No03: NOP   0;
NoXX: NOP   0;
NETWORK
TITLE =ASW_6030: Active step germinating
//      U     "MAL1S021Par".Par.FlagProcess.ProcessActive;
//      SPBN  tuen;
//
//// copy stepnr
//      L     "MAL1S021Par".Par.ParIntMachine.ActualStep;
//      T     "MAL1S021Par".Par.ParIntProcess.ActualStep;
//// set step conditions
//
//// Case where process is starting during loading
//      U     "MAL1S021Par".Par.FlagProcess.ProcessActive;
//      UN    "MAL1S021Par".Par.FlagFunction_1.StepLoading; // Step loading
//      SPBN  e003;
//// lifting devices must be in highest position
//      L       WinCoS_BIW01_09PLC1BIW01_02.Ma.Par.ParPositionTopRightUnits;
////Malting Plant OAO Belsolod Ivanonvo Weissrussland
//      L     50; // 50mm offset
//      +I    ;
//      T     "MAL1S021Par".Par.MachineValue.SOLLWERT_HUBZUG1_HOEHE;
//      L       WinCoS_BIW01_09PLC1BIW01_02.Ma.Par.ParPositionTopLeftUnits;
////Malting Plant OAO Belsolod Ivanonvo Weissrussland
//      L     50; // 50mm offset
//      +I    ;
//      T     "MAL1S021Par".Par.MachineValue.SOLLWERT_HUBZUG2_HOEHE;
//      L     5;
//      T     WinCoS_BIW01_09PLC1BIW01_02.Ma.Par.ParTolPosition;
//e003: NOP   0;
//
//// reset turning cmds
//
//// save turning cmds from prev.step
//      L     "MAL1S021Par".Par.ParIntMachine.ActualStep;
//      L     "MAL1S021Par".Par.ParIntProcess.PrevStep1stTurn;
//      <>I   ;
//      SPB   sav1;
//      U     "MAL1S021Par".Par.FlagProcess2.Turning1WithSpraying;
//      =     "MAL1S021Par".Par.Switches1.StaOn08; // Turning1WithSpraying
//      U     "MAL1S021Par".Par.FlagProcess2.Turning1WithDosing;
//      =     "MAL1S021Par".Par.Switches1.StaOn09; // Turning1WithDosing
//sav1: NOP   0;
//      L     "MAL1S021Par".Par.ParIntMachine.ActualStep;
//      L     "MAL1S021Par".Par.ParIntProcess.PrevStep2ndTurn;
//      <>I   ;
//      SPB   sav2;
//      U     "MAL1S021Par".Par.FlagProcess2.Turning2WithSpraying;
//      =     "MAL1S021Par".Par.Switches1.StaOn10; // Turning2WithSpraying
//      U     "MAL1S021Par".Par.FlagProcess2.Turning2WithDosing;
//      =     "MAL1S021Par".Par.Switches1.StaOn11; // Turning2WithDosing
//sav2: NOP   0;
//
//      SET   ;
//      R     "MAL1S021Par".Par.FlagProcess2.Turning1WithoutSpraying;
//      R     "MAL1S021Par".Par.FlagProcess2.Turning1WithSpraying;
//      R     "MAL1S021Par".Par.FlagProcess2.Turning1WithDosing;
//      R     "MAL1S021Par".Par.FlagProcess2.Turning2WithoutSpraying;
//      R     "MAL1S021Par".Par.FlagProcess2.Turning2WithSpraying;
//      R     "MAL1S021Par".Par.FlagProcess2.Turning2WithDosing;
//
//// Delta Temp to switch to next step
//      L     "MAL1S021Par".StepAct.DeltaTempSwitchpointStep;
//      L     L#0;
//      >D   ;
//      =     "MAL1S021Par".Par.FlagProcess1.DeltaTempNextStep;
//// Max Temp to switch to next step
//      L     "MAL1S021Par".StepAct.MaxTempAboveFloorStep;
//      L     L#0;
//      >D   ;
//      =     "MAL1S021Par".Par.FlagProcess1.MaxTempNextStep;
//
//// position waste air see sub 6050
//
//// basic speed fan see sub 6040
//
//// air humifidication
//      L     1;
//      L     "MAL1S021Par".StepAct.AirMoisten;   // On/Off
//      ==I;  // air humifidication on
//      U     WinCoS_BIW01_09PLC1BIW01_02.Ma.StStartedFwd; //Malting Plant OAO Be
//lsolod Ivanonvo Weissrussland
//      =     "MAL1S021Par".Par.FlagProcess.AirHumidificationValve1; // air humif
//idication valve 1 on
//      U(    ; // air humifidication on
//      L     "MAL1S021Par".Par.ParIntMachine.TargetSpeedGermFan; // germinating
//fan is running
//      L     40; // fanspeed > 40%
//      >I    ; // muss noch in Istwert getauscht werden JV
//      )     ; // fanspeed > 40%
//      =     "MAL1S021Par".Par.FlagProcess.AirHumidificationValve2;
//
//// air cooling
//      L     "MAL1S021Par".StepAct.Cooling;
//      L   1;  // Activate Cooling System = 1 (yes)
//      ==I;
//      =     "MAL1S021Par".Par.FlagProcess.Cooling; // request cooling
//
//      U     "MAL1S021Par".Par.FlagProcess.ProcessActive;
//      U     "MAL1S021".PCRead.Step.StReady;
//      UN    "MAL1S021Par".Par.FlagFunction_1.StepLoading;
//      SPBN  e630;
//
//// turning 1
//      UN    "MAL1S021Par".Par.FlagProcess2.StartSecondTurningRound; // Turn
//from PrevStep
//      U(;
//      L     "MAL1S021Par".StepAct.StartTurningRound_1;
//      L     0;
//      >=D;                  // negative, no turning 1
//      );
//      U(    ;
//      O(    ; // Nach Rezept
//      L     "MAL1S021Par".ActTimeStepProcess.StepTimeActHourTotal; // Steptime
//in hours overall
//      L     "MAL1S021Par".StepAct.StartTurningRound_1;
//      ==I   ;
//      UN     WinCoS_BIW01_09PLC1BIW01_02.Ma.StAdjusted; // target position
//turning reached
//      )     ;
//      O(    ; // Selbsthaltung
//      L     "MAL1S021Par".ActTimeStepProcess.StepTimeActHourTotal; // Steptime i
//n hours overall
//      L     "MAL1S021Par".StepAct.StartTurningRound_1;
//      <>I   ;
//      U     "MAL1S021Par".Par.FlagProcess2.StartFirstTurningRound;
//      )     ;
//      )     ;
//      S     "MAL1S021Par".Par.FlagProcess2.Turning1WithoutSpraying;
//      S     "MAL1S021Par".Par.FlagFunction_1.TurningStart;
//// turning 1 with spraying
//      U(    ;
//      L     1;
//      L     "MAL1S021Par".StepAct.TurningWithSpraying_1;
//      ==I;    // turning 1 with spraying on
//      U(    ;
//      L     "MAL1S021Par".Par.ParIntMachine.ActualStep;
//      L     "MAL1S021Par".Par.ParIntProcess.PrevStep1stTurn;
//      ==I   ;
//      )     ;
//      )     ;
//      O(    ;
//      L     "MAL1S021Par".Par.ParIntMachine.ActualStep;
//      L     "MAL1S021Par".Par.ParIntProcess.PrevStep1stTurn;
//      <>I   ;
//      U     "MAL1S021Par".Par.Switches1.StaOn08; // Turning1WithSpraying
//      )     ;
//      U     "MAL1S021Par".Par.FlagProcess2.Turning1WithoutSpraying;
//      S     "MAL1S021Par".Par.FlagProcess2.Turning1WithSpraying;
//// turning 1 with spraying and GA3
//      U(    ;
//      L     1;
//      L     "MAL1S021Par".StepAct.TurningWithDosing_1;
//      ==I;    // turning 1 with spraying on
//      U(    ;
//      L     "MAL1S021Par".Par.ParIntMachine.ActualStep;
//      L     "MAL1S021Par".Par.ParIntProcess.PrevStep1stTurn;
//      ==I   ;
//      )     ;
//      )     ;
//      O(    ;
//      L     "MAL1S021Par".Par.ParIntMachine.ActualStep;
//      L     "MAL1S021Par".Par.ParIntProcess.PrevStep1stTurn;
//      <>I   ;
//      U     "MAL1S021Par".Par.Switches1.StaOn09; // Turning1WithDosing
//      )     ;
//      U     "MAL1S021Par".Par.FlagProcess2.Turning1WithoutSpraying;
//      S     "MAL1S021Par".Par.FlagProcess2.Turning1WithSpraying;
//      S     "MAL1S021Par".Par.FlagProcess2.Turning1WithDosing;
//
//      U     "MAL1S021Par".Par.FlagProcess2.Turning1WithoutSpraying;
//      U     "MAL1S021Par".Par.FlagFunction_1.TurningStart;
//      UN     WinCoS_BIW01_09PLC1BIW01_02.Ma.StAdjusted; // target position turni
//ng reached
//      FP    "MAL1S021Par".Par.FlagProcess2.StartFirstTurningFP;
//      S     "MAL1S021Par".Par.FlagProcess2.StartFirstTurningRound;
//
//      U     WinCoS_BIW01_09PLC1BIW01_02.Ma.StAdjusted; // target position
//turning reached
//      O(    ;
//      L     "MAL1S021Par".ActTimeStepProcess.StepTimeActHourTotal; // Steptime i
//n hours overall
//      L     "MAL1S021Par".StepAct.StartTurningRound_1;
//      >I    ;
//      U     WinCoS_BIW01_09PLC1BIW01_02.Ma.StAdjusted; // target position
//turning reached
//      )     ;
//      U     "MAL1S021Par".Par.FlagProcess2.StartFirstTurningRound;
//      R     "MAL1S021Par".Par.FlagProcess2.StartFirstTurningRound;
//
//      U     "MAL1S021Par".Par.FlagProcess2.StartFirstTurningFP;
//      SPB   trn1;
//      L     "MAL1S021Par".Par.ParIntMachine.ActualStep;
//      T     "MAL1S021Par".Par.ParIntProcess.PrevStep1stTurn;
//trn1: NOP   0;
//
//// turning 2
//      UN    "MAL1S021Par".Par.FlagProcess2.StartFirstTurningRound; // Unsinngie
//Rezeptwerte
//      U(;
//      L     1;
//      L     "MAL1S021Par".StepAct.StartTurningRound_2;
//      ==I    ;
//      );
//      U(    ;
//      O(    ; // Nach Rezept
//      L     "MAL1S021Par".ActTimeStepProcess.StepTimeActHourTotal; // Steptime i
//n hours overall
//      L     "MAL1S021Par".StepAct.StartTurningRound_2;
//      ==I   ;
//      UN     WinCoS_BIW01_09PLC1BIW01_02.Ma.StAdjusted; // target position
//turning reached
//      )     ;
//      O(    ; // Selbsthaltung
//      L     "MAL1S021Par".ActTimeStepProcess.StepTimeActHourTotal; // Steptime
//in hours overall
//      L     "MAL1S021Par".StepAct.StartTurningRound_2;
//      <>I   ;
//      U     "MAL1S021Par".Par.FlagProcess2.StartSecondTurningRound;
//      )     ;
//      )     ;
//      S     "MAL1S021Par".Par.FlagProcess2.Turning2WithoutSpraying;
//      S     "MAL1S021Par".Par.FlagFunction_1.TurningStart;
//// turning 2 with spraying
//      U(    ;
//      L     1;
//      L     "MAL1S021Par".StepAct.TurningWithSpraying_2;
//      ==I    ;
//      U(    ;
//      L     "MAL1S021Par".Par.ParIntMachine.ActualStep;
//      L     "MAL1S021Par".Par.ParIntProcess.PrevStep2ndTurn;
//      ==I   ;
//      )     ;
//      )     ;
//      O(    ;
//      L     "MAL1S021Par".Par.ParIntMachine.ActualStep;
//      L     "MAL1S021Par".Par.ParIntProcess.PrevStep2ndTurn;
//      <>I   ;
//      U     "MAL1S021Par".Par.Switches1.StaOn10; // Turning2WithSpraying
//      )     ;
//      U     "MAL1S021Par".Par.FlagProcess2.Turning2WithoutSpraying;
//      S     "MAL1S021Par".Par.FlagProcess2.Turning2WithSpraying;
//// turning 2 with spraying and GA3
//      U(    ;
//      L     1;
//      L     "MAL1S021Par".StepAct.TurningWithDosing_2;
//      ==I;    // turning 2 with spraying and GA3 on
//      U(    ;
//      L     "MAL1S021Par".Par.ParIntMachine.ActualStep;
//      L     "MAL1S021Par".Par.ParIntProcess.PrevStep2ndTurn;
//      ==I   ;
//      )     ;
//      )     ;
//      O(    ;
//      L     "MAL1S021Par".Par.ParIntMachine.ActualStep;
//      L     "MAL1S021Par".Par.ParIntProcess.PrevStep2ndTurn;
//      <>I   ;
//      U     "MAL1S021Par".Par.Switches1.StaOn11; // Turning2WithDosing
//      )     ;
//      U     "MAL1S021Par".Par.FlagProcess2.Turning2WithoutSpraying;
//      S     "MAL1S021Par".Par.FlagProcess2.Turning2WithSpraying;
//      S     "MAL1S021Par".Par.FlagProcess2.Turning2WithDosing;
//
//      U     "MAL1S021Par".Par.FlagProcess2.Turning2WithoutSpraying;
//      U     "MAL1S021Par".Par.FlagFunction_1.TurningStart;
//      UN     WinCoS_BIW01_09PLC1BIW01_02.Ma.StAdjusted; // target position
//turning reached
//      FP    "MAL1S021Par".Par.FlagProcess2.StartSecondTurningFP;
//      S     "MAL1S021Par".Par.FlagProcess2.StartSecondTurningRound;
//
//      U     WinCoS_BIW01_09PLC1BIW01_02.Ma.StAdjusted; // target position
//turning reached
//      O(    ;
//      L     "MAL1S021Par".ActTimeStepProcess.StepTimeActHourTotal; // Steptime
//in hours overall
//      L     "MAL1S021Par".StepAct.StartTurningRound_2;
//      >I    ;
//      U     WinCoS_BIW01_09PLC1BIW01_02.Ma.StAdjusted; // target position
//turning reached
//      )     ;
//      U     "MAL1S021Par".Par.FlagProcess2.StartSecondTurningRound;
//      R     "MAL1S021Par".Par.FlagProcess2.StartSecondTurningRound;
//
//      U     "MAL1S021Par".Par.FlagProcess2.StartSecondTurningFP;
//      SPB   trn2;
//      L     "MAL1S021Par".Par.ParIntMachine.ActualStep;
//      T     "MAL1S021Par".Par.ParIntProcess.PrevStep2ndTurn;
//trn2: NOP   0;
////Fix Speed for Turning
//      U     "MAL1S021Par".Par.FlagProcess2.Turning1WithoutSpraying;
//      O     "MAL1S021Par".Par.FlagProcess2.Turning1WithSpraying;
//      O     "MAL1S021Par".Par.FlagProcess2.Turning2WithoutSpraying;
//      O     "MAL1S021Par".Par.FlagProcess2.Turning2WithSpraying;
//      U    M 50.0;
//      SPBN  SpdT;
//      L     15; // 15Hz
//      T     "MAL1S021Par".Par.MachineValue.SollwertFahrantrieb;
//SpdT: NOP   0;
//
//// find turning direction
//      U     "MAL1S021Par".Par.FlagGen.TurningStarted;
//      O(    ;
//      UN    "MAL1S021Par".Par.FlagProcess2.Turning1WithoutSpraying;
//      UN    "MAL1S021Par".Par.FlagProcess2.Turning2WithoutSpraying;
//      )     ;
//      SPB   tuen;
//      L     "MAL1S021Par".Par.ParIntMachine.TargetPosTravDriTurnRigt; // 370° =
//endposition turning right
//      T     WinCoS_BIW01_09PLC1BIW01_02.Ma.InPositionTarget; // target position
//turning reached
//
//      U(    ;
//      L     WinCoS_BIW01_09PLC1BIW01_02.Ma.OutPositionAngle;
//      L     1800;
//      <I    ; // condition turning right (clockwise)
//      )     ;
//      S     "MAL1S021Par".Par.FlagFunction_1.TurningRight;
//      S     "MAL1S021Par".Par.FlagGen.TurningStarted;
//// - Correct effect of ILO Mode
//      L       WinCoS_BIW01_09PLC1BIW01_02.Ma.Par.ParPositionTopLeftUnits; //Malt
//ing Plant OAO Belsolod Ivanonvo Weissrussland
//      T     "MAL1S021Par".Par.MachineValue.SOLLWERT_HUBZUG1_HOEHE;
//      L       WinCoS_BIW01_09PLC1BIW01_02.Ma.Par.ParPositionTopRightUnits; //Mal
//ting Plant OAO Belsolod Ivanonvo Weissrussland
//      T     "MAL1S021Par".Par.MachineValue.SOLLWERT_HUBZUG2_HOEHE;
//      SPB   E603   ;
//      L     "MAL1S021Par".Par.ParIntMachine.TargetPosTravDriTurnLeft; // 0° =
//endposition turning left
//      T     WinCoS_BIW01_09PLC1BIW01_02.Ma.InPositionTarget; // target position
//turning reached
//
//      U(    ;
//      L     WinCoS_BIW01_09PLC1BIW01_02.Ma.OutPositionAngle;
//      L     1800;
//      >=I   ; // condition turning left (counterclockwise)
//      )     ;
//      S     "MAL1S021Par".Par.FlagFunction_1.TurningLeft;
//      S     "MAL1S021Par".Par.FlagGen.TurningStarted;
//// - Correct effect of ILO Mode
//      L       WinCoS_BIW01_09PLC1BIW01_02.Ma.Par.ParPositionTopLeftUnits;
////Malting Plant OAO Belsolod Ivanonvo Weissrussland
//      T     "MAL1S021Par".Par.MachineValue.SOLLWERT_HUBZUG1_HOEHE;
//      L       WinCoS_BIW01_09PLC1BIW01_02.Ma.Par.ParPositionTopRightUnits;
////Malting Plant OAO Belsolod Ivanonvo Weissrussland
//      T     "MAL1S021Par".Par.MachineValue.SOLLWERT_HUBZUG2_HOEHE;
//      SPB   E603   ;
//tuen: NOP   0;
//// - Case of fast speed to protect a 2nd start during same hours as finsihed
//      O(    ; // Nach Rezept
//      L     "MAL1S021Par".ActTimeStepProcess.StepTimeActHourTotal; // Steptime i
//n hours overall
//      L     "MAL1S021Par".StepAct.StartTurningRound_1;
//      ==I   ;
//      U     WinCoS_BIW01_09PLC1BIW01_02.Ma.StAdjusted; // target position turnin
//g reached
//      U     "MAL1S021Par".Par.FlagFunction_1.TurningStart;
//      )     ;
//      O(    ; // Nach Rezept
//      L     "MAL1S021Par".ActTimeStepProcess.StepTimeActHourTotal; // Steptime i
//n hours overall
//      L     "MAL1S021Par".StepAct.StartTurningRound_2;
//      ==I   ;
//      U     WinCoS_BIW01_09PLC1BIW01_02.Ma.StAdjusted; // target position
//turning reached
//      U     "MAL1S021Par".Par.FlagFunction_1.TurningStart;
//      )     ;
//      SPB   e603;
//
//// reset turning right (clockwise)
//      U     "MAL1S021Par".Par.FlagFunction_1.TurningRight;
//      U(    ;
//      O      WinCoS_BIW01_09PLC1BIW01_02.Ma.StAdjusted; // target position
//turning reached
//      O(    ;
//      L     WinCoS_BIW01_09PLC1BIW01_02.Ma.OutPositionAngle;
//      L     WinCoS_BIW01_09PLC1BIW01_02.Ma.Par.ParTolPosition;
//      +I    ;
//      L     "MAL1S021Par".Par.ParIntMachine.TargetPosTravDriTurnRigt;
//      >=I   ;
//      )     ;
//      )     ;
//      R     "MAL1S021Par".Par.FlagFunction_1.TurningRight;
//      R     "MAL1S021Par".Par.FlagFunction_1.TurningStart;
//
//// reset turning left (counterclockwise)
//      U     "MAL1S021Par".Par.FlagFunction_1.TurningLeft;
//      U(    ;
//      O     WinCoS_BIW01_09PLC1BIW01_02.Ma.StAdjusted; // target position turnin
//g reached
//      O(    ;
//      L     WinCoS_BIW01_09PLC1BIW01_02.Ma.OutPositionAngle;
//      L     WinCoS_BIW01_09PLC1BIW01_02.Ma.Par.ParTolPosition;
//      -I    ;
//      L     "MAL1S021Par".Par.ParIntMachine.TargetPosTravDriTurnLeft;
//      <=I   ;
//      )     ;
//      )     ;
//      R     "MAL1S021Par".Par.FlagFunction_1.TurningLeft;
//      R     "MAL1S021Par".Par.FlagFunction_1.TurningStart;
//
//// reset turning flag
//      U     "MAL1S021Par".Par.FlagGen.TurningStarted;
//      UN    "MAL1S021Par".Par.FlagProcess2.Turning1WithoutSpraying;
//      UN    "MAL1S021Par".Par.FlagProcess2.Turning2WithoutSpraying;
//      O(    ;
//      U     "MAL1S021Par".Par.FlagGen.TurningStarted;
//      U     WinCoS_BIW01_09PLC1BIW01_02.Ma.StAdjusted; // target position
//turning reached
//      )     ;
//      ON    "MAL1S021Par".Par.FlagProcess.ProcessActive;
//      R     "MAL1S021Par".Par.FlagGen.TurningStarted;
//      R     "MAL1S021Par".Par.FlagProcess2.Turning1WithoutSpraying;
//      R     "MAL1S021Par".Par.FlagProcess2.Turning2WithoutSpraying;
//      R     "MAL1S021Par".Par.FlagFunction_1.TurningStart;
//e630: NOP   0;
//      UN    "MAL1S021Par".Par.FlagProcess.ProcessActive;
//      R     "MAL1S021Par".Par.FlagProcess2.StartFirstTurningRound;
//      R     "MAL1S021Par".Par.FlagProcess2.StartSecondTurningRound;
//
//e603: NOP   0;
//E603: NOP   0;



      U     "MAL1S021Par".Par.FlagProcess.ProcessActive;
      SPBN  tuen;

// copy stepnr
      L     "MAL1S021Par".Par.ParIntMachine.ActualStep;
      T     "MAL1S021Par".Par.ParIntProcess.ActualStep;
// set step conditions

// reset turning cmds

// save turning cmds from prev.step
      L     "MAL1S021Par".Par.ParIntMachine.ActualStep;
      L     "MAL1S021Par".Par.ParIntProcess.PrevStep1stTurn;
      <>I   ;
      SPB   sav1;
      U     "MAL1S021Par".Par.FlagProcess2.Turning1WithSpraying;
      =     "MAL1S021Par".Par.Switches1.StaOn08; // Turning1WithSpraying
      U     "MAL1S021Par".Par.FlagProcess2.Turning1WithDosing;
      =     "MAL1S021Par".Par.Switches1.StaOn09; // Turning1WithDosing
sav1: NOP   0;
      L     "MAL1S021Par".Par.ParIntMachine.ActualStep;
      L     "MAL1S021Par".Par.ParIntProcess.PrevStep2ndTurn;
      <>I   ;
      SPB   sav2;
      U     "MAL1S021Par".Par.FlagProcess2.Turning2WithSpraying;
      =     "MAL1S021Par".Par.Switches1.StaOn10; // Turning2WithSpraying
      U     "MAL1S021Par".Par.FlagProcess2.Turning2WithDosing;
      =     "MAL1S021Par".Par.Switches1.StaOn11; // Turning2WithDosing
sav2: NOP   0;

      SET   ;
      R     "MAL1S021Par".Par.FlagProcess2.Turning1WithoutSpraying;
      R     "MAL1S021Par".Par.FlagProcess2.Turning1WithSpraying;
      R     "MAL1S021Par".Par.FlagProcess2.Turning1WithDosing;
      R     "MAL1S021Par".Par.FlagProcess2.Turning2WithoutSpraying;
      R     "MAL1S021Par".Par.FlagProcess2.Turning2WithSpraying;
      R     "MAL1S021Par".Par.FlagProcess2.Turning2WithDosing;

// Delta Temp to switch to next step
      L     "MAL1S021Par".StepAct.DeltaTempSwitchpointStep;
      L     L#0;
      >D    ;
      =     "MAL1S021Par".Par.FlagProcess1.DeltaTempNextStep;
// Max Temp to switch to next step
      L     "MAL1S021Par".StepAct.MaxTempAboveFloorStep;
      L     L#0;
      >D    ;
      =     "MAL1S021Par".Par.FlagProcess1.MaxTempNextStep;

// position waste air see sub 6050

// basic speed fan see sub 6040

// air humifidication

// air cooling
      L     "MAL1S021Par".StepAct.Cooling;
      L     1; // Activate Cooling System = 1 (yes)
      ==I   ;
      =     "MAL1S021Par".Par.FlagProcess.Cooling; // request cooling

      U     "MAL1S021Par".Par.FlagProcess.ProcessActive;
      U     "MAL1S021".PCRead.Step.StReady;
      UN    "MAL1S021Par".Par.FlagFunction_1.StepLoading;
      SPBN  e630;

// turning 1
      UN    "MAL1S021Par".Par.FlagProcess2.StartSecondTurningRound; // Turn from PrevStep
      U(    ;
      L     "MAL1S021Par".StepAct.StartTurningRound_1;
      L     0;
      >=I   ; // negative, no turning 1
      )     ;
      U(    ;
      O(    ; // Nach Rezept
      L     "MAL1S021Par".ActTimeStepProcess.StepTimeActHourTotal; // Steptime in hours overall
      L     "MAL1S021Par".StepAct.StartTurningRound_1;
      ==I   ;
      UN    "G185M".A_2511_MXZ41MA.Ma.StAdjusted; // target position turning reached
      )     ;
      O(    ; // Selbsthaltung
      L     "MAL1S021Par".ActTimeStepProcess.StepTimeActHourTotal; // Steptime in hours overall
      L     "MAL1S021Par".StepAct.StartTurningRound_1;
      <>I   ;
      U     "MAL1S021Par".Par.FlagProcess2.StartFirstTurningRound;
      )     ;
      )     ;
      S     "MAL1S021Par".Par.FlagProcess2.Turning1WithoutSpraying;
      S     "MAL1S021Par".Par.FlagFunction_1.TurningStart;
// turning 1 with spraying
      U(    ;
      L     1;
      L     "MAL1S021Par".StepAct.TurningWithSpraying_1;
      ==I   ; // turning 1 with spraying on
      U(    ;
      L     "MAL1S021Par".Par.ParIntMachine.ActualStep;
      L     "MAL1S021Par".Par.ParIntProcess.PrevStep1stTurn;
      ==I   ;
      )     ;
      )     ;
      O(    ;
      L     "MAL1S021Par".Par.ParIntMachine.ActualStep;
      L     "MAL1S021Par".Par.ParIntProcess.PrevStep1stTurn;
      <>I   ;
      U     "MAL1S021Par".Par.Switches1.StaOn08; // Turning1WithSpraying
      )     ;
      U     "MAL1S021Par".Par.FlagProcess2.Turning1WithoutSpraying;
      S     "MAL1S021Par".Par.FlagProcess2.Turning1WithSpraying;
// turning 1 with spraying and GA3
      U(    ;
      L     1;
      L     "MAL1S021Par".StepAct.TurningWithDosing_1;
      ==I   ; // turning 1 with spraying on
      U(    ;
      L     "MAL1S021Par".Par.ParIntMachine.ActualStep;
      L     "MAL1S021Par".Par.ParIntProcess.PrevStep1stTurn;
      ==I   ;
      )     ;
      )     ;
      O(    ;
      L     "MAL1S021Par".Par.ParIntMachine.ActualStep;
      L     "MAL1S021Par".Par.ParIntProcess.PrevStep1stTurn;
      <>I   ;
      U     "MAL1S021Par".Par.Switches1.StaOn09; // Turning1WithDosing
      )     ;
      U     "MAL1S021Par".Par.FlagProcess2.Turning1WithoutSpraying;
      S     "MAL1S021Par".Par.FlagProcess2.Turning1WithSpraying;
      S     "MAL1S021Par".Par.FlagProcess2.Turning1WithDosing;

//BRT070410 - wird einen Zyklus später gesetzt
      U     "MAL1S021Par".Par.FlagProcess2.StartFirstDosingFP;
      S     "MAL1S021Par".Par.FlagProcess2.StartFirstTurningRound;

      U     "MAL1S021Par".Par.FlagProcess2.Turning1WithoutSpraying;
      U     "MAL1S021Par".Par.FlagFunction_1.TurningStart;
//BRT140310      UN    "G185M".A_2511_MXZ41MA.Ma.StAdjusted    // target position turning reached
      UN    "G185M".A_2511_MXZ41MA.Ma.OutAdjusted; // target position turning reached
      FP    "MAL1S021Par".Par.FlagProcess2.StartFirstTurningFP;
      =     "MAL1S021Par".Par.FlagProcess2.StartFirstDosingFP;
//BRT070410      S     "MAL1S021Par".Par.FlagProcess2.StartFirstTurningRound

      U     "MAL1S021Par".Par.FlagProcess2.StartFirstDosingFP;
      U     "MAL1S021Par".Par.FlagProcess2.StartFirstTurningFP;
      SPBN  trn1;
      L     "MAL1S021Par".Par.ParIntMachine.ActualStep;
      T     "MAL1S021Par".Par.ParIntProcess.PrevStep1stTurn;
trn1: NOP   0;

//BRT140310      U     "G185M".A_2511_MXZ41MA.Ma.StAdjusted    // target position turning reached
      U     "G185M".A_2511_MXZ41MA.Ma.OutAdjusted; // target position turning reached
      O(    ;
      L     "MAL1S021Par".ActTimeStepProcess.StepTimeActHourTotal; // Steptime in hours overall
      L     "MAL1S021Par".StepAct.StartTurningRound_1;
      >I    ;
      U(    ;
      O     "G185M".A_2511_MXZ41MA.Ma.OutAdjusted; // target position turning reached
      O(    ;
//BRT140310      UN    "G185M".A_2511_BZS46.StTrue // stop fan side
//BRT140310      U     "G185M".A_2511_BZS44.StTrue // stop discharge side
      U     "G185M".A_2511_BZS46.StTrue; // stop fan side
      UN    "G185M".A_2511_BZS44.StTrue; // stop discharge side
      U     "MAL1S021Par".Par.FlagFunction_1.TurningRight;
      )     ;
      O(    ;
//BRT140310      U     "G185M".A_2511_BZS46.StTrue // stop fan side
//BRT140310      UN    "G185M".A_2511_BZS44.StTrue // stop discharge side
      UN    "G185M".A_2511_BZS46.StTrue; // stop fan side
      U     "G185M".A_2511_BZS44.StTrue; // stop discharge side
      U     "MAL1S021Par".Par.FlagFunction_1.TurningLeft;
      )     ;
      )     ;
      )     ;
      O(    ;
      L     "MAL1S021Par".StepAct.StartTurningRound_1;
//BRT140310      L     0
//BRT140310      <D                                // negative, no turning 1
      L     -1; //BRT140310
      ==I   ; //BRT140310
      )     ;
      U     "MAL1S021Par".Par.FlagProcess2.StartFirstTurningRound;
      R     "MAL1S021Par".Par.FlagProcess2.StartFirstTurningRound;
      R     "MAL1S021Par".Par.Switches1.StaOn08; // Turning1WithSpraying
      R     "MAL1S021Par".Par.Switches1.StaOn09; // Turning1WithDosing

// turning 2
      UN    "MAL1S021Par".Par.FlagProcess2.StartFirstTurningRound; // Unsinnige Rezeptwerte
      U(    ;
//BRT160310      L     1
      L     "MAL1S021Par".StepAct.StartTurningRound_2;
      L     0; //BRT160310
      >=I   ;
      )     ;
      U(    ;
      O(    ; // Nach Rezept
      L     "MAL1S021Par".ActTimeStepProcess.StepTimeActHourTotal; // Steptime in hours overall
      L     "MAL1S021Par".StepAct.StartTurningRound_2;
      ==I   ;
      UN    "G185M".A_2511_MXZ41MA.Ma.StAdjusted; // target position turning reached
      )     ;
      O(    ; // Selbsthaltung
      L     "MAL1S021Par".ActTimeStepProcess.StepTimeActHourTotal; // Steptime in hours overall
      L     "MAL1S021Par".StepAct.StartTurningRound_2;
      <>I   ;
      U     "MAL1S021Par".Par.FlagProcess2.StartSecondTurningRound;
      )     ;
      )     ;
      S     "MAL1S021Par".Par.FlagProcess2.Turning2WithoutSpraying;
      S     "MAL1S021Par".Par.FlagFunction_1.TurningStart;
// turning 2 with spraying
      U(    ;
      L     1;
      L     "MAL1S021Par".StepAct.TurningWithSpraying_2;
      ==I   ;
      U(    ;
      L     "MAL1S021Par".Par.ParIntMachine.ActualStep;
      L     "MAL1S021Par".Par.ParIntProcess.PrevStep2ndTurn;
      ==I   ;
      )     ;
      )     ;
      O(    ;
      L     "MAL1S021Par".Par.ParIntMachine.ActualStep;
      L     "MAL1S021Par".Par.ParIntProcess.PrevStep2ndTurn;
      <>I   ;
      U     "MAL1S021Par".Par.Switches1.StaOn10; // Turning2WithSpraying
      )     ;
      U     "MAL1S021Par".Par.FlagProcess2.Turning2WithoutSpraying;
      S     "MAL1S021Par".Par.FlagProcess2.Turning2WithSpraying;
// turning 2 with spraying and GA3
      U(    ;
      L     1;
      L     "MAL1S021Par".StepAct.TurningWithDosing_2;
      ==I   ; // turning 2 with spraying and GA3 on
      U(    ;
      L     "MAL1S021Par".Par.ParIntMachine.ActualStep;
      L     "MAL1S021Par".Par.ParIntProcess.PrevStep2ndTurn;
      ==I   ;
      )     ;
      )     ;
      O(    ;
      L     "MAL1S021Par".Par.ParIntMachine.ActualStep;
      L     "MAL1S021Par".Par.ParIntProcess.PrevStep2ndTurn;
      <>I   ;
      U     "MAL1S021Par".Par.Switches1.StaOn11; // Turning2WithDosing
      )     ;
      U     "MAL1S021Par".Par.FlagProcess2.Turning2WithoutSpraying;
      S     "MAL1S021Par".Par.FlagProcess2.Turning2WithSpraying;
      S     "MAL1S021Par".Par.FlagProcess2.Turning2WithDosing;

//BRT070410 - wird einen Zyklus später gesetzt
      U     "MAL1S021Par".Par.FlagProcess2.StartSecondDosingFP;
      S     "MAL1S021Par".Par.FlagProcess2.StartSecondTurningRound;

      U     "MAL1S021Par".Par.FlagProcess2.Turning2WithoutSpraying;
      U     "MAL1S021Par".Par.FlagFunction_1.TurningStart;
//BRT140310      UN    "G185M".A_2511_MXZ41MA.Ma.StAdjusted    // target position turning reached
      UN    "G185M".A_2511_MXZ41MA.Ma.OutAdjusted; // target position turning reached
      FP    "MAL1S021Par".Par.FlagProcess2.StartSecondTurningFP;
      =     "MAL1S021Par".Par.FlagProcess2.StartSecondDosingFP;
//BRT070410      S     "MAL1S021Par".Par.FlagProcess2.StartSecondTurningRound

      U     "MAL1S021Par".Par.FlagProcess2.StartSecondDosingFP;
      U     "MAL1S021Par".Par.FlagProcess2.StartSecondTurningFP;
      SPBN  trn2;
      L     "MAL1S021Par".Par.ParIntMachine.ActualStep;
      T     "MAL1S021Par".Par.ParIntProcess.PrevStep2ndTurn;
trn2: NOP   0;

//BRT140310      U     "G185M".A_2511_MXZ41MA.Ma.StAdjusted    // target position turning reached
      U     "G185M".A_2511_MXZ41MA.Ma.OutAdjusted; // target position turning reached
      O(    ;
      L     "MAL1S021Par".ActTimeStepProcess.StepTimeActHourTotal; // Steptime in hours overall
      L     "MAL1S021Par".StepAct.StartTurningRound_2;
      >I    ;
      U(    ;
      O     "G185M".A_2511_MXZ41MA.Ma.OutAdjusted; // target position turning reached
      O(    ;
      UN    "G185M".A_2511_BZS46.StTrue; // stop fan side
      U     "G185M".A_2511_BZS44.StTrue; // stop discharge side
      U     "MAL1S021Par".Par.FlagFunction_1.TurningRight;
      )     ;
      O(    ;
      U     "G185M".A_2511_BZS46.StTrue; // stop fan side
      UN    "G185M".A_2511_BZS44.StTrue; // stop discharge side
      U     "MAL1S021Par".Par.FlagFunction_1.TurningLeft;
      )     ;
      )     ;
      )     ;
      O(    ;
      L     "MAL1S021Par".StepAct.StartTurningRound_2;
//BRT140310      L     0
//BRT140310      <D                                // negative, no turning 1
      L     -1; //BRT140310
      ==I   ; //BRT140310
      )     ;
      U     "MAL1S021Par".Par.FlagProcess2.StartSecondTurningRound;
      R     "MAL1S021Par".Par.FlagProcess2.StartSecondTurningRound;
      R     "MAL1S021Par".Par.Switches1.StaOn10; // Turning2WithSpraying
      R     "MAL1S021Par".Par.Switches1.StaOn11; // Turning2WithDosing

      L     3600;
      T     "MAL1S021Par".Par.ParIntMachine.TargetPosTravDriTurnRigt; // 360° = endposition turning right

// find turning direction spez. APU: right ==> forward, left ==> reverse
      U     "MAL1S021Par".Par.FlagGen.TurningStarted;
      O(    ;
      UN    "MAL1S021Par".Par.FlagProcess2.Turning1WithoutSpraying;
      UN    "MAL1S021Par".Par.FlagProcess2.Turning2WithoutSpraying;
      )     ;
      SPB   tuen;
      L     "MAL1S021Par".Par.ParIntMachine.TargetPosTravDriTurnRigt; // 360° = endposition turning right
      T     "G185M".A_2511_MXZ41MA.Ma.InPositionTarget; // target position turning

      U(    ;
      L     "G185M".A_2511_MXZ41MA.Ma.OutPositionAngle;
      L     1800;
      <I    ; // condition turning right (clockwise)
      )     ;
//BRT140310      O     "G185M".A_2511_BZS46.StTrue // stop fan side
//BRT140310      UN    "G185M".A_2511_BZS44.StTrue // stop discharge side
      O     "G185M".A_2511_BZS44.StTrue; // stop zeroposition  //BRT070310
      UN    "G185M".A_2511_BZS46.StTrue; //stop end side   //BRT070310
      S     "MAL1S021Par".Par.FlagFunction_1.TurningRight;
      S     "MAL1S021Par".Par.FlagGen.TurningStarted;
      SPB   E603;
      L     "MAL1S021Par".Par.ParIntMachine.TargetPosTravDriTurnLeft; // 0° = endposition turning left
      T     "G185M".A_2511_MXZ41MA.Ma.InPositionTarget; // target position turning

      U(    ;
      L     "G185M".A_2511_MXZ41MA.Ma.OutPositionAngle;
      L     1800;
      >=I   ; // condition turning left (counterclockwise)
      )     ;
//BRT140310      O     "G185M".A_2511_BZS44.StTrue // stop discharge side
//BRT140310      UN    "G185M".A_2511_BZS46.StTrue // stop fan side
      O     "G185M".A_2511_BZS46.StTrue; // stop zeroposition  //BRT070310
      UN    "G185M".A_2511_BZS44.StTrue; //stop end side   //BRT070310
      S     "MAL1S021Par".Par.FlagFunction_1.TurningLeft;
      S     "MAL1S021Par".Par.FlagGen.TurningStarted;
      SPB   E603;
tuen: NOP   0;

// reset turning right (clockwise)
      U     "MAL1S021Par".Par.FlagFunction_1.TurningRight;
      U(    ;
//      O     "G202M"._2111_MXZ41MA.Ma.StAdjusted    // target position turning reached
      O(    ;
      L     "G185M".A_2511_MXZ41MA.Ma.OutPositionAngle;
      L     "G185M".A_2511_MXZ41MA.Ma.Par.ParTolPosition;
      +I    ;
      L     "MAL1S021Par".Par.ParIntMachine.TargetPosTravDriTurnRigt;
      >=I   ;
      )     ;
//BRT140310      O     "G185M".A_2511_BZS44.StTrue // stop discharge side
      O     "G185M".A_2511_BZS46.StTrue; // stop zeroposition
      )     ;
      R     "MAL1S021Par".Par.FlagFunction_1.TurningRight;
      R     "MAL1S021Par".Par.FlagFunction_1.TurningStart;

// reset turning left (counterclockwise)
      U     "MAL1S021Par".Par.FlagFunction_1.TurningLeft;
      U(    ;
//      O     "G202M"._2111_MXZ41MA.Ma.StAdjusted    // target position turning reached
      O(    ;
      L     "G185M".A_2511_MXZ41MA.Ma.OutPositionAngle;
      L     "G185M".A_2511_MXZ41MA.Ma.Par.ParTolPosition;
      -I    ;
      L     "MAL1S021Par".Par.ParIntMachine.TargetPosTravDriTurnLeft;
      <=I   ;
      )     ;
      O     "G185M".A_2511_BZS44.StTrue; // stop end side
//BRT140310      O     "G185M".A_2511_BZS46.StTrue // stop fan side
      )     ;
      R     "MAL1S021Par".Par.FlagFunction_1.TurningLeft;
      R     "MAL1S021Par".Par.FlagFunction_1.TurningStart;

// - Case of fast speed to protect a 2nd start during same hours as finsihed
      U     "MAL1S021Par".Par.FlagGen.TurningStarted;
//====>BRT140310      UN    "MAL1S021Par".Par.FlagProcess.ProcessEnd    // JV210808 to finish last turning
      U(    ;
      U     "MAL1S021Par".Par.FlagProcess2.Turning1WithoutSpraying;
      O     "MAL1S021Par".Par.FlagProcess2.Turning2WithoutSpraying;
      UN    "MAL1S021Par".Par.FlagProcess.ProcessEnd; // JV210808 to finish last turning
      )     ;
      UN    "MAL1S021StepValues".StartStep; // start step for average calculating
      U(    ;
      O(    ; // Nach Rezept
      U(    ;
      L     "MAL1S021Par".ActTimeStepProcess.StepTimeActHourTotal; // Steptime in hours overall
      L     "MAL1S021Par".StepAct.StartTurningRound_1;
      ==I   ; // JV 250808
      )     ;
//      UN    "MAL1S021Par".Par.FlagProcess2.StartFirstTurningRound    // JV 250808
      U     "G185M".A_2511_MXZ41MA.Ma.OutAdjusted; // target position turning reached
      )     ;
      O(    ; // Nach Rezept
      U(    ;
      L     "MAL1S021Par".ActTimeStepProcess.StepTimeActHourTotal; // Steptime in hours overall
      L     "MAL1S021Par".StepAct.StartTurningRound_2;
      ==I   ; // JV 250808
      )     ;
//      UN    "MAL1S021Par".Par.FlagProcess2.StartSecondTurningRound    // JV 250808
      U     "G185M".A_2511_MXZ41MA.Ma.OutAdjusted; // target position turning reached
//<====BRT140310
      )     ;
      )     ;
      O(    ;
      UN    "G185M".A_2511_MXZ41MA.Ma.OutAdjusted; // target position turning reached
      UN    "MAL1S021Par".Par.FlagFunction_1.StepUnloading;
      )     ;
      SPB   e603;

// reset turning flag
      U     "MAL1S021Par".Par.FlagGen.TurningStarted;
      ON    "MAL1S021Par".Par.FlagProcess.ProcessActive;
      R     "MAL1S021Par".Par.FlagGen.TurningStarted;
      R     "MAL1S021Par".Par.FlagProcess2.Turning1WithoutSpraying;
      R     "MAL1S021Par".Par.FlagProcess2.Turning2WithoutSpraying;
      R     "MAL1S021Par".Par.FlagProcess2.Turning1WithSpraying;
      R     "MAL1S021Par".Par.FlagProcess2.Turning2WithSpraying;
      R     "MAL1S021Par".Par.FlagProcess2.Turning1WithDosing;
      R     "MAL1S021Par".Par.FlagProcess2.Turning2WithDosing;
      R     "MAL1S021Par".Par.FlagFunction_1.TurningStart;
      R     "MAL1S021Par".Par.FlagProcess2.StartFirstTurningRound; // JV 250808
      R     "MAL1S021Par".Par.FlagProcess2.StartSecondTurningRound; // JV 250808
      SET   ;
      R     "MAL1S021StepValues".StartStep; // start step for average calculating
e630: NOP   0;
      UN    "MAL1S021Par".Par.FlagProcess.ProcessActive;
      R     "MAL1S021Par".Par.FlagProcess2.StartFirstTurningRound;
      R     "MAL1S021Par".Par.FlagProcess2.StartSecondTurningRound;
      R     "MAL1S021Par".Par.Switches1.StaOn08; // Turning1WithSpraying
      R     "MAL1S021Par".Par.Switches1.StaOn09; // Turning1WithDosing
      R     "MAL1S021Par".Par.Switches1.StaOn10; // Turning2WithSpraying
      R     "MAL1S021Par".Par.Switches1.StaOn11; // Turning2WithDosing

      L     "G185M".A_2511_MXZ41MA.Ma.OutPositionAngle;
      T     "G185M".A_2511_MXZ41MA.Ma.OutPositionAngle;

      L     "G185M".A_2511_MXZ41MA.Ma.OutPositionRel;
      T     "G185M".A_2511_MXZ41MA.Ma.OutPositionRel;

e603: NOP   0;
E603: NOP   0;


NETWORK
TITLE =ASW_6040: Set fanspeed by delta-t
//Die Drehzahl des Ventilators wird zwischen dem Rezeptsollwert, als Untere
//Grenze, und 100% oder Rezeptsollwert, als obere Grenze, geregelt. Die Regelung
//erfolgt nach folgendem Prinzip:
//"Delta-T" ist die Differenz zwischen der Soll-Temperatur (Rezeptsollwert) unter
//der Horde und der gemessenen Ist-Temperatur über der Horde.
//Steigt die Ist-Temperatur über der Horde und "Delta-T" wird > als der Sollwert
//im Rezept, so wird die Drehzahl des Ventilators stufenweise erhöht. Maximale
//Drehzahl ist 100% oder Rezeptsollwert.
//Sinkt die Ist-Temperatur über der Horde und "Delta-T" wird < als der Sollwert
//im
//Rezept, so wird die Drehzahl des Ventilators stufenweise verringert. Minimale
//Drehzahl ist der Rezeptsollwert.
//Die Rampen (Stufen) werden durch den Technologen festgelegt und in Programmcode
//eingetragen. Es sind keine Rezeptsollwerte.
      NOP   0;
//====>BRT140310
// recipe setpoint
//      L     "MAL1S021Par".StepAct.SpeedVentilatorBasic
//      L     0
//      ==I                               // no fan during turning
//      SPB   e604                        // JV040908
      UN(   ;
      U(    ;
      L     "MAL1S021Par".Par.ParIntMachine.ActualStep;
      L     1;
      ==I   ;
      )     ;
      UN(   ;
      L     "MAL1S021Par".Par.ProcessValue.StepTimeAct; // in ms
      L     L#1000; // in first secunde steptime
      >D    ;
      )     ;
      )     ;
// BRT140310 - berechneter Targetwert darf nur bei StepNr.1 oder! Rezeptwert-Änderung überschrieben werden
      U(    ;
      L     "MAL1S021Par".StepAct.SpeedVentilatorBasic;
      L     "MAL1S021Par".Par.ParIntProcess.Value23; // Rezeptwert vor Änderung
      ==D   ;
      )     ;
      SPB   regu;
      L     "MAL1S021Par".StepAct.SpeedVentilatorBasic;
      T     "MAL1S021Par".Par.ParIntProcess.Value23; // Rezeptwert vor Änderung
      SPA   Summ;
regu: NOP   0;

// BRT140310 - nicht nötig, da obige Änderung bei Änderung Rezeptwert (Modify) auch Target-Wert neu lädt
//      U     "MAL1S019".ToASW.CmdModify
//      SPB   Summ
//<====BRT140310


// Setpoint
      L     "MAL1S021Par".StepAct.TemperaturAboveFloor;
      L     "MAL1S021Par".StepAct.TemperaturBelowFloor;
      -D    ;
      T     "MAL1S021Par".Par.ProcessValue.SetpointDeltaTempDint;
// actual value
      L     "G188M".A_2591_BTE02.OutValueUnits; //AIR TEMPERATURE ABOVE FLOOR
      L     "G188M".A_2591_BTE01.OutValueUnits; //AIR TEMPERATURE BELOW FLOOR
      -D    ;
      L     L#10; //BRT140310
      /D    ; //BRT140310
      T     "MAL1S021Par".Par.ProcessValue.ActValueDeltaTempDint;
// flags to inc/dec
      L     "MAL1S021Par".Par.ProcessValue.SetpointDeltaTempDint;
      -D    ;
      T     "MAL1S021Par".Par.ProcessValue.ResultDeltaTemp;
      L     L#0;
      >D    ;
      =     "MAL1S021Par".Par.FlagProcess1.DeltaTempPlus;
      <D    ;
      =     "MAL1S021Par".Par.FlagProcess1.DeltaTempMinus;

      U     "MAL1S021Par".Par.FlagProcess1.DeltaTempPlus;
//BRT200310      U     "SYS_Scan0_Tick1min"
      U     "SYS_Scan0_Tick30s"; //Scan0_Tick30s
      SPBN  dec;
      L     "MAL1S021Par".Par.ParIntMachine.TargetSpeedGermFan;
      L     100; // linmit max
      >=I   ;
      O(    ; //JV160710 =====>
      TAK   ;
      L     "MAL1S021Par".StepAct.SpeedVentilatorMaximal;
      >=I   ;
      U(    ;
      L     "MAL1S021Par".StepAct.SpeedVentilatorMaximal;
      L     "MAL1S021Par".StepAct.SpeedVentilatorBasic;
      >=I   ;
      )     ;
      )     ; //JV160710 <=====
      SPB   dec;
      L     "MAL1S021Par".Par.ParIntMachine.TargetSpeedGermFan;
      L     1;
      +I    ;
      T     "MAL1S021Par".Par.ParIntMachine.TargetSpeedGermFan;
      SPA   e604;
dec:  NOP   0;
      U     "MAL1S021Par".Par.FlagProcess1.DeltaTempMinus;
      O(    ; //JV160710 =====>
      L     "MAL1S021Par".Par.ParIntMachine.TargetSpeedGermFan;
      L     "MAL1S021Par".StepAct.SpeedVentilatorMaximal;
      >I    ;
      )     ; //JV160710 <=====
//BRT200310      U     "SYS_Scan0_Tick1min"
      U     "SYS_Scan0_Tick30s"; //Scan0_Tick30s
      SPBN  e604;
      L     "MAL1S021Par".Par.ParIntMachine.TargetSpeedGermFan;
      L     "MAL1S021Par".StepAct.SpeedVentilatorBasic; // linmit min
      <=I   ;
      SPB   e604;
      L     "MAL1S021Par".Par.ParIntMachine.TargetSpeedGermFan;
      L     1;
      -I    ;
      T     "MAL1S021Par".Par.ParIntMachine.TargetSpeedGermFan;
      SPA   e604;

Summ: NOP   0;
      L     "MAL1S021Par".StepAct.SpeedVentilatorBasic;
      T     "MAL1S021Par".Par.ParIntMachine.TargetSpeedGermFan;
      U     "MAL1S021Par".Par.FlagProcess.ProcessEnd; // JV030908
      UN    "MAL1S021".PCRead.Step.StEmptying;
      UN    "MAL1S021".PCRead.Step.StEmptied;
      SPBN  e604;
      L     "MAL1S021Par".Par.ParIntProcess.SavedTargetSpeedGermFan;
      T     "MAL1S021Par".Par.ParIntMachine.TargetSpeedGermFan;
e604: NOP   0;
// store actual setpoint
      U     "MAL1S021Par".Par.FlagProcess.ProcessActive;
      U(    ;
      L     "MAL1S021Par".StepAct.SpeedVentilatorBasic;
      L     0; // setpoint recipe > 0
      >I    ;
      )     ;
      SPBN  E604;
      L     "MAL1S021Par".StepAct.SpeedVentilatorBasic;
      T     "MAL1S021Par".Par.ParIntProcess.SavedTargetSpeedGermFan;
E604: NOP   0;
//-------------------------------------------------------------------------------------------------
//--- Ventilator 2 einzeln geregelt ---
      UN(   ;
      U(    ;
      L     "MAL1S021Par".Par.ParIntMachine.ActualStep;
      L     1;
      ==I   ;
      )     ;
      UN(   ;
      L     "MAL1S021Par".Par.ProcessValue.StepTimeAct; // in ms
      L     L#1000; // in first secunde steptime
      >D    ;
      )     ;
      )     ;
// BRT040310 - berechneter Targetwert darf nur bei StepNr.1 oder! Rezeptwert-Änderung überschrieben werden
      U(    ;
      L     "MAL1S021Par".StepAct.SpeedVentilatorBasic;
      L     "MAL1S021Par".Par.ParIntProcess.Value25; // Rezeptwert vor Änderung
      ==D   ;
      )     ;
      SPB   reg1;
      L     "MAL1S021Par".StepAct.SpeedVentilatorBasic;
      T     "MAL1S021Par".Par.ParIntProcess.Value25; // Rezeptwert vor Änderung
      SPA   Sum1;
reg1: NOP   0;
// Setpoint
      L     "MAL1S021Par".StepAct.TemperaturAboveFloor;
      L     "MAL1S021Par".StepAct.TemperaturBelowFloor;
      -D    ;
      T     "MAL1S021Par".Par.ProcessValue.Value13; // Setpoint Delta Temp
// actual value
      L     "G188M".A_2591_BTE04.OutValueUnits; //AIR TEMPERATURE ABOVE FLOOR
      L     "G188M".A_2591_BTE03.OutValueUnits; //AIR TEMPERATURE BELOW FLOOR
      -D    ;
      L     L#10; //BRT060310
      /D    ; //BRT060310
      T     "MAL1S021Par".Par.ProcessValue.Value14; // Actual Value Delta Temp
// flags to inc/dec
      L     "MAL1S021Par".Par.ProcessValue.Value13; // Setpoint Delta Temp
      -D    ;
      T     "MAL1S021Par".Par.ProcessValue.Value15; // Result Delta Temp
      L     L#0;
      >D    ;
      =     "MAL1S021Par".Par.FlagProcess1.Inf23; // Delta Temp Plus
      <D    ;
      =     "MAL1S021Par".Par.FlagProcess1.Inf24; // Delta Temp Minus

      U     "MAL1S021Par".Par.FlagProcess1.Inf23; // Delta Temp Plus
//BRT203010      U     "SYS_Scan0_Tick1min"
      U     "SYS_Scan0_Tick30s"; //Scan0_Tick30s
      SPBN  dec1;
      L     "MAL1S021Par".Par.ParIntProcess.Value26; // Target Speed GermFan 2
      L     100; // linmit max
      >=I   ;
      O(    ; //JV160710 =====>
      TAK   ;
      L     "MAL1S021Par".StepAct.SpeedVentilatorMaximal;
      >=I   ;
      U(    ;
      L     "MAL1S021Par".StepAct.SpeedVentilatorMaximal;
      L     "MAL1S021Par".StepAct.SpeedVentilatorBasic;
      >=I   ;
      )     ;
      )     ; //JV160710 <=====
      SPB   dec1;
      L     "MAL1S021Par".Par.ParIntProcess.Value26; // Target Speed GermFan 2
      L     1;
      +I    ;
      T     "MAL1S021Par".Par.ParIntProcess.Value26; // Target Speed GermFan 2
      SPA   e614;
dec1: NOP   0;
      U     "MAL1S021Par".Par.FlagProcess1.Inf24; // Delta Temp Minus
      O(    ; //JV160710 =====>
      L     "MAL1S021Par".Par.ParIntProcess.Value26; // Target Speed GermFan 2
      L     "MAL1S021Par".StepAct.SpeedVentilatorMaximal;
      >I    ;
      )     ; //JV160710 <=====
//BRT200310      U     "SYS_Scan0_Tick1min"
      U     "SYS_Scan0_Tick30s"; //Scan0_Tick30s
      SPBN  e614;
      L     "MAL1S021Par".Par.ParIntProcess.Value26; // Target Speed GermFan 2
      L     "MAL1S021Par".StepAct.SpeedVentilatorBasic; // linmit min
      <=I   ;
      SPB   e614;
      L     "MAL1S021Par".Par.ParIntProcess.Value26; // Target Speed GermFan 2
      L     1;
      -I    ;
      T     "MAL1S021Par".Par.ParIntProcess.Value26; // Target Speed GermFan 2
      SPA   e614;

Sum1: NOP   0;
      L     "MAL1S021Par".StepAct.SpeedVentilatorBasic;
      T     "MAL1S021Par".Par.ParIntProcess.Value26; // Target Speed GermFan 2
      U     "MAL1S021Par".Par.FlagProcess.ProcessEnd; // JV030908
      UN    "MAL1S021".PCRead.Step.StEmptying;
      UN    "MAL1S021".PCRead.Step.StEmptied;
      SPBN  e614;
      L     "MAL1S021Par".Par.ParIntProcess.Value27; // Saved Target Speed GermFan 2
      T     "MAL1S021Par".Par.ParIntProcess.Value26; // Target Speed GermFan 2
e614: NOP   0;
// store actual setpoint
      U     "MAL1S021Par".Par.FlagProcess.ProcessActive;
      U(    ;
      L     "MAL1S021Par".StepAct.SpeedVentilatorBasic;
      L     0; // setpoint recipe > 0
      >I    ;
      )     ;
      SPBN  E614;
      L     "MAL1S021Par".StepAct.SpeedVentilatorBasic;
      T     "MAL1S021Par".Par.ParIntProcess.Value27; // Saved Target Speed GermFan 2
E614: NOP   0;

NETWORK
TITLE =ASW_6050: Position waste air
//Der Betriebsart Sommerbetrieb/Winterbetrieb wird durch den Bediener per Rezept
//bestimmt.
//Wird die Kühlung im Rezept angewählt, so erfolgt die Umschaltung AUF
//Sommerbetrieb. Die Frischluftklappe wird nach dem Rezeptsollwert gestellt.
//Es erfolgt keine Regelung.
//Wird die Kühlung im Rezept abgewählt, so erfolgt die Umschaltung AUF
//Winterbetrieb. Die Frischluftklappe wird zuerst nach dem Rezeptsollwert
//gestellt. Der Rezeptsollwert ist die untere Grenze für die Regelung.
//Wird die Soll-Temperatur unter der Horde von Kühl- Heizanlage nicht eingehalten
//-Temperatur zu hoch und der Schaltpunkt überschritten, so wird die
//Frischluftklappe stufenweise geöffnet.
//Maximalwert ist 100%.
//Wird die Soll-Temperatur unter der Horde von Kühl- Heizanlage nicht eingehalten
//-Temperatur zu niedrig und der Schaltpunkt unterschritten, so wird die
//Frischluftklappe stufenweise geschlossen.
//Minimalwert ist der Rezeptsollwert.
//-------------------------------------------------------------------------------
//      NOP   0
//// setpoint waste air                    = 100% - setpoint fresh air
//      L     100
//      L     "MAL1S021Par".StepAct.PosFreshAirFlapBasic
//      -I
//      T     "MAL1S021Par".StepAct.PosWasteAirFlapBasic
//
//// setpoint limit maximal position fresh air
//      L     100
//      T     "MAL1S021Par".StepAct.PosFreshAirFlapMax    // limit max
//      L     L#10                        // 1,0°
//      T     "MAL1S021Par".StepAct.DeltaTempSwitchpointAir
//
//// recipe setpoint
//      L     "MAL1S021Par".Par.ProcessValue.StepTimeAct    // in ms
//      L     L#1000                      // in first secunde steptime
//      >D
//      SPB   Reg
//      SPA   summ
//Reg:  NOP   0
//
//// Cooling or heating from cooling defive active --> no flap regulation!
////      U     "ENG_RemarkFlag"
////      U     "ComDB_Cooling".Ma.ACK.ActivFlag.Cool.Germinating_1_Started //
//Internal or external coooling is running
////      O     "MAL1S017".ToASW.CmdModify
////      SPB   summ
//
////Conditions to activate cooling -- With flap regulation
//      U(
//      L     1
//      L     "MAL1S021Par".StepAct.Cooling    // On/Off
//      ==I                               // Cooling on
//      U     "MAL1S021Par".Par.FlagProcess.ProcessActive
//      )
//      U     "G190M".A_2560_MXZ01.StStartedFwd
//      U     "G190M".A_2560_MXZ02.StStartedFwd
//      U(
//      L     "G269M".A_3191_BTE11.OutValueUnits    //WET BULB TEMPERATURE OUTSIDE
//      L     20                          // 2,0°C Hysteresis
//      -D
//      L     "MAL1S021Par".StepAct.TemperaturBelowFloor    //SET POINT
//TEMPERATURE RECIPE
//      >=D
//      )
//      U(
//      L     "G188M".A_2591_BTE01.OutValueUnits    //AIR TEMPERATURE BELOW FLOOR
//GM2
//      L     10                          // 1,0°C Hysteresis
//      -D
//      L     "MAL1S021Par".StepAct.TemperaturBelowFloor    //SET POINT
//TEMPERATURE RECIPE
//      >=D
//      )
//      U(
//      L     "G188M".A_2591_BTE02.OutValueUnits    //AIR TEMPERATURE ABOVE FLOOR
//GM2
//      L     20                          // 2,0°C Hysteresis
//      -D
//      L     "MAL1S021Par".StepAct.TemperaturBelowFloor    //SET POINT
//TEMPERATURE RECIPE
//      >=D
//      )
//      S     "MAL1S021Par".Par.FlagProcess.Cooling_Activ
//
//      U(
//      L     0
//      L     "MAL1S021Par".StepAct.Cooling    // On/Off
//      ==I                               // Cooling off
//      )
//      ON    "G190M".A_2560_MXZ01.StStartedFwd
//      ON    "G190M".A_2560_MXZ02.StStartedFwd
//      O(
//      L     "G269M".A_3191_BTE11.OutValueUnits    //WET BULB TEMPERATURE OUTSIDE
//      L     10                          // 1,0°C Hysteresis
//      +D
//      L     "MAL1S021Par".StepAct.TemperaturBelowFloor    //SET POINT
//TEMPERATURE RECIPE
//      <D
//      )
//      O(
//      L     "G188M".A_2591_BTE02.OutValueUnits    //AIR TEMPERATURE ABOVE FLOOR
//GM1
//      L     10                          // 1,0°C Hysteresis
//      +D
//      L     "MAL1S021Par".StepAct.TemperaturBelowFloor    //SET POINT
//TEMPERATURE RECIPE
//      <D
//      )
//      R     "MAL1S021Par".Par.FlagProcess.Cooling_Activ
//
//      U     "MAL1S021Par".Par.FlagProcess.Cooling_Activ
//      SPB   summ
//
//// Check the minimum opening of fresh air louver
//      U(
//      L     "MAL1S021Par".Par.ParIntMachine.TargetPosFreshAir
//      L     "MAL1S021Par".StepAct.PosFreshAirFlapBasic
//      <I
//      )
//      SPBN  modi
//      L     "MAL1S021Par".StepAct.PosFreshAirFlapBasic    //Basic position %
//      T     "MAL1S021Par".Par.ParIntMachine.TargetPosFreshAir
//modi: NOP   0
//
////-Recipe modify-
//      U(                                // Nach gesundem Menschenverstand
//      L     "MAL1S021Par".StepAct.PosFreshAirFlapBasic
//      L     "MAL1S021Par".Par.ParIntMachine.TargetPosFreshAir
//      >I
//      U     "MAL1S021Par".Par.FlagProcess1.FreshAirFlapOPEN
//      )
//      O(                                // Nach gesundem Menschenverstand
//      L     "MAL1S021Par".StepAct.PosFreshAirFlapBasic
//      L     "MAL1S021Par".Par.ParIntMachine.TargetPosFreshAir
//      <I
//      U     "MAL1S021Par".Par.FlagProcess1.FreshAirFlapCLOSE
//      )
//      O(                                // Nach gesundem Menschenverstand
//      L     "MAL1S021Par".StepAct.PosFreshAirFlapBasic
//      L     "MAL1S021Par".Par.ParIntMachine.TargetPosFreshAir
//      <>I
//      UN    "MAL1S021Par".Par.FlagProcess1.FreshAirFlapOPEN
//      UN    "MAL1S021Par".Par.FlagProcess1.FreshAirFlapCLOSE
//      )
//      O(                                // 1. Versuch den Technologen ruhig
//stellen
//      L     "MAL1S021Par".StepAct.PosFreshAirFlapBasic
//      L     "MAL1S021Par".Par.ParIntProcess.SavedTargetPosFreshAir
//      <>I
//      )
//      U     "MAL1S021".ToASW.CmdModify
//      SPB   summ
////      L     "G168M".A_2491_BTE01.OutValueUnits    //AIR TEMPERATURE BELOW
//FLOOR
////      L     L#10                        // von xx,xx°C AUF xx,x°C
////      /D
////      L     "MAL1S017Par".StepAct.TemperaturBelowFloor
////      -D
////      L     "MAL1S017Par".StepAct.DeltaTempSwitchpointAir
////      >D
////      =     "MAL1S017Par".Par.FlagProcess1.FreshAirFlapOPEN
//
////      L     "G128M".A_2191_BTE01.OutValueUnits    //AIR TEMPERATURE BELOW
//FLOOR
////      L     L#10                        // von xxx,xx°C AUF xxx,x°C
////      /D
////      L     "MAL1S017Par".StepAct.TemperaturBelowFloor
////      TAK
////      -D
////      L     "MAL1S017Par".StepAct.DeltaTempSwitchpointAir
////      >D
////      =     "MAL1S017Par".Par.FlagProcess1.FreshAirFlapCLOSE
//      U(
//      L     "G188M".A_2591_BTE01.OutValueUnits    //AIR TEMPERATURE BELOW FLOOR
//GM1
//      L     "MAL1S021Par".StepAct.TemperaturBelowFloor    //SET POINT
//TEMPERATURE RECIPE
//      <D
//      )
//      U(
//      L     "G269M".A_3191_BTE11.OutValueUnits    //WET BULB TEMPERATURE OUTSIDE
//      L     "G188M".A_2591_BTE02.OutValueUnits    //AIR TEMPERATURE ABOVE FLOOR
//GM1
//      >D
//      )
//      O
//      U(
//      L     "G188M".A_2591_BTE01.OutValueUnits    //AIR TEMPERATURE BELOW FLOOR
//GM1
//      L     "MAL1S021Par".StepAct.TemperaturBelowFloor    //SET POINT
//TEMPERATURE RECIPE
//      >D
//      )
//      U(
//      L     "G269M".A_3191_BTE11.OutValueUnits    //WET BULB TEMPERATURE OUTSIDE
//      L     "G188M".A_2591_BTE01.OutValueUnits    //AIR TEMPERATURE BELOW FLOOR
//GM1
//      <D
//      )
//      =     "MAL1S021Par".Par.FlagProcess1.FreshAirFlapOPEN
//
//      U(
//      L     "G188M".A_2591_BTE01.OutValueUnits    //AIR TEMPERATURE BELOW FLOOR
//GM1
//      L     "MAL1S021Par".StepAct.TemperaturBelowFloor    //SET POINT
//TEMPERATURE RECIPE
//      <D
//      )
//      U(
//      L     "G269M".A_3191_BTE11.OutValueUnits    //WET BULB TEMPERATURE OUTSIDE
//      L     "G188M".A_2591_BTE02.OutValueUnits    //AIR TEMPERATURE ABOVE FLOOR
//GM1
//      <D
//      )
//      =     "MAL1S021Par".Par.FlagProcess1.FreshAirFlapCLOSE
//
//      U     "MAL1S021Par".Par.FlagProcess1.FreshAirFlapOPEN
//      U     "SYS_Scan0_Tick1min"
//      SPBN  dez
//      L     "MAL1S021Par".Par.ParIntMachine.TargetPosWasteAir
//      L     100                         // limit max
//      >=I
//      SPB   dez
//      L     "MAL1S021Par".Par.ParIntMachine.TargetPosWasteAir
//      L     1
//      +I
//      T     "MAL1S021Par".Par.ParIntMachine.TargetPosWasteAir
//      SPA   e605
//dez:  NOP   0
//      U     "MAL1S021Par".Par.FlagProcess1.FreshAirFlapCLOSE
//      U     "SYS_Scan0_Tick1min"
//      SPBN  e605
//      L     "MAL1S021Par".Par.ParIntMachine.TargetPosWasteAir
//      L     "MAL1S021Par".StepAct.PosFreshAirFlapBasic    // limit min
//      <=I
//      SPB   e605
//      L     "MAL1S021Par".Par.ParIntMachine.TargetPosWasteAir
//      L     1
//      -I
//      T     "MAL1S021Par".Par.ParIntMachine.TargetPosWasteAir
//      SPA   e605
//
//summ: NOP   0
//      U     "G269M".read_3191
//      SPBN  bypa
//      U(
//      L     "G188M".A_2591_BTE02.OutValueUnits    //AIR TEMPERATURE ABOVE FLOOR
//GM1
//      L     10                          // 1,0°C Hysteresis
//      -D
//      L     "G269M".A_3191_BTE11.OutValueUnits    //WET BULB TEMPERATURE OUTSIDE
//      >=D
//      )
//      SPB   tar1
//      U(
//      L     "G188M".A_2591_BTE02.OutValueUnits    //AIR TEMPERATURE ABOVE FLOOR
//GM1
//      L     10                          // 1,0°C Hysteresis
//      +D
//      L     "G269M".A_3191_BTE11.OutValueUnits    //WET BULB TEMPERATURE OUTSIDE
//      <=D
//      )
//      SPB   tar0
//      SPA   bypa
//tar1: L     100                         //open fresh air 100%
//      T     "MAL1S021Par".Par.ParIntMachine.TargetPosFreshAir
//      SPA   bypa
//tar0: L     "MAL1S021Par".StepAct.PosFreshAirFlapBasic    //close fresh air to
//Basic position %
//      T     "MAL1S021Par".Par.ParIntMachine.TargetPosFreshAir
//bypa: NOP   0
////************************************************************************
//      U     "MAL1S021Par".Par.FlagProcess.ProcessEnd    // JV030908
//      UN    "MAL1S021".PCRead.Step.StEmptying
//      UN    "MAL1S021".PCRead.Step.StEmptied    // JV030908
//      SPBN  e605
//      L     "MAL1S021Par".Par.ParIntProcess.SavedTargetPosFreshAir
//      T     "MAL1S021Par".Par.ParIntMachine.TargetPosFreshAir
//e605: NOP   0
//      L     100
//      L     "MAL1S021Par".Par.ParIntMachine.TargetPosFreshAir
//      -I
//      T     "MAL1S021Par".Par.ParIntMachine.TargetPosWasteAir
//// store actual setpoint
//      U     "MAL1S021Par".Par.FlagProcess.ProcessActive
//      U(
//      L     "MAL1S021Par".StepAct.PosFreshAirFlapBasic
//      L     0                           // setpoint recipe > 0
//      >I
//      )
//      SPBN  E605
//      L     "MAL1S021Par".StepAct.PosFreshAirFlapBasic
//      T     "MAL1S021Par".Par.ParIntProcess.SavedTargetPosFreshAir
//E605: NOP   0
//
//BRT140310 - keine AMBEV Steuerung!!!
      NOP   0;
// setpoint limit maximal position fresh air
      L     100;
      T     "MAL1S021Par".StepAct.PosFreshAirFlapMax; // limit max
      L     L#5; // 0,5°
      T     "MAL1S021Par".StepAct.DeltaTempSwitchpointAir;

// recipe setpoint
      UN(   ;
      U(    ;
      L     "MAL1S021Par".Par.ParIntMachine.ActualStep;
      L     1;
      ==I   ;
      )     ;
      UN(   ;
      L     "MAL1S021Par".Par.ProcessValue.StepTimeAct; // in ms
      L     L#1000; // in first secunde steptime
      >D    ;
      )     ;
      )     ;
// BRT17102009 - berechneter Targetwert darf nur bei StepNr.1 oder! Rezeptwert-Änderung überschrieben werden
      U(    ;
      L     "MAL1S021Par".StepAct.PosFreshAirFlapBasic;
      L     "MAL1S021Par".Par.ParIntProcess.Value24; // Rezeptwert vor Änderung
      ==D   ;
      )     ;
      SPB   Reg;
      L     "MAL1S021Par".StepAct.PosFreshAirFlapBasic;
      T     "MAL1S021Par".Par.ParIntProcess.Value24; // Rezeptwert vor Änderung

      L     "MAL1S021Par".StepAct.PosFreshAirFlapBasic;
      T     "MAL1S021Par".Par.ParIntMachine.TargetPosFreshAir;
      SPA   e605;
Reg:  NOP   0;

// Cooling or heating from cooling defive active --> no flap regulation!
//BRT140310 - Cooling angewählt in Rezept!
      U     "MAL1S021Par".Par.FlagProcess.Cooling; // request cooling
      SPB   summ;

      L     "G188M".A_2591_BTE01.OutValueUnits; //AIR TEMPERATURE BELOW FLOOR
      L     L#10; // von xx,xx°C AUF xx,x°C
      /D    ;
      L     "MAL1S021Par".StepAct.TemperaturBelowFloor;
      -D    ;
      L     "MAL1S021Par".StepAct.DeltaTempSwitchpointAir;
      >D    ;
      =     "MAL1S021Par".Par.FlagProcess1.FreshAirFlapOPEN;

      L     "G188M".A_2591_BTE01.OutValueUnits; //AIR TEMPERATURE BELOW FLOOR
      L     L#10; // von xxx,xx°C AUF xxx,x°C
      /D    ;
      L     "MAL1S021Par".StepAct.TemperaturBelowFloor;
      TAK   ;
      -D    ;
      L     "MAL1S021Par".StepAct.DeltaTempSwitchpointAir;
      >D    ;
      =     "MAL1S021Par".Par.FlagProcess1.FreshAirFlapCLOSE;

      U     "MAL1S021Par".Par.FlagProcess1.FreshAirFlapOPEN;
      U     "SYS_Scan0_Tick1min";
      SPBN  dez;
      L     "MAL1S021Par".Par.ParIntMachine.TargetPosFreshAir;
      L     "MAL1S021Par".StepAct.PosFreshAirFlapMax; // limit max
      >=I   ;
      SPB   dez;
      L     "MAL1S021Par".Par.ParIntMachine.TargetPosFreshAir;
      L     1;
      +I    ;
      T     "MAL1S021Par".Par.ParIntMachine.TargetPosFreshAir;
      SPA   e605;
dez:  NOP   0;
      U     "MAL1S021Par".Par.FlagProcess1.FreshAirFlapCLOSE;
      U     "SYS_Scan0_Tick1min";
      SPBN  e605;
      L     "MAL1S021Par".Par.ParIntMachine.TargetPosFreshAir;
      L     "MAL1S021Par".StepAct.PosFreshAirFlapBasic; // limit min
      <=I   ;
      SPB   e605;
      L     "MAL1S021Par".Par.ParIntMachine.TargetPosFreshAir;
      L     1;
      -I    ;
      T     "MAL1S021Par".Par.ParIntMachine.TargetPosFreshAir;
      SPA   e605;

summ: NOP   0;
      L     "MAL1S021Par".StepAct.PosFreshAirFlapBasic;
      T     "MAL1S021Par".Par.ParIntMachine.TargetPosFreshAir;
      SPA   e605;

e605: NOP   0;
//------------------------------------------------------------------------------------------------
//--- Position Fresh-/Recycling-Air Flap 2 ---
// recipe setpoint
      UN(   ;
      U(    ;
      L     "MAL1S021Par".Par.ParIntMachine.ActualStep;
      L     1;
      ==I   ;
      )     ;
      UN(   ;
      L     "MAL1S021Par".Par.ProcessValue.StepTimeAct; // in ms
      L     L#1000; // in first secunde steptime
      >D    ;
      )     ;
      )     ;
// BRT17102009 - berechneter Targetwert darf nur bei StepNr.1 oder! Rezeptwert-Änderung überschrieben werden
      U(    ;
      L     "MAL1S021Par".StepAct.PosFreshAirFlapBasic;
      L     "MAL1S021Par".Par.ParIntProcess.Value28; // Rezeptwert vor Änderung
      ==D   ;
      )     ;
      SPB   Reg1;
      L     "MAL1S021Par".StepAct.PosFreshAirFlapBasic;
      T     "MAL1S021Par".Par.ParIntProcess.Value28; // Rezeptwert vor Änderung

      L     "MAL1S021Par".StepAct.PosFreshAirFlapBasic;
      T     "MAL1S021Par".Par.ParIntProcess.Value29; // Target Position FreshAir 2
      SPA   e615;
Reg1: NOP   0;

// Cooling or heating from cooling defive active --> no flap regulation!
//BRT030310 - Cooling angewählt in Rezept!
      U     "MAL1S021Par".Par.FlagProcess.Cooling; // request cooling
      SPB   sum1;

      L     "G188M".A_2591_BTE03.OutValueUnits; //AIR TEMPERATURE BELOW FLOOR
      L     L#10; // von xx,xx°C AUF xx,x°C
      /D    ;
      L     "MAL1S021Par".StepAct.TemperaturBelowFloor;
      -D    ;
      L     "MAL1S021Par".StepAct.DeltaTempSwitchpointAir;
      >D    ;
      =     "MAL1S021Par".Par.FlagProcess.Inf05; // FreshAir Flap OPEN

      L     "G188M".A_2591_BTE03.OutValueUnits; //AIR TEMPERATURE BELOW FLOOR
      L     L#10; // von xxx,xx°C AUF xxx,x°C
      /D    ;
      L     "MAL1S021Par".StepAct.TemperaturBelowFloor;
      TAK   ;
      -D    ;
      L     "MAL1S021Par".StepAct.DeltaTempSwitchpointAir;
      >D    ;
      =     "MAL1S021Par".Par.FlagProcess.Inf06; // FreshAir Flap CLOSE

      U     "MAL1S021Par".Par.FlagProcess.Inf05; // FreshAir Flap OPEN
      U     "SYS_Scan0_Tick1min";
      SPBN  dez1;
      L     "MAL1S021Par".Par.ParIntProcess.Value29; // Target Position FreshAir 2
      L     "MAL1S021Par".StepAct.PosFreshAirFlapMax; // limit max
      >=I   ;
      SPB   dez1;
      L     "MAL1S021Par".Par.ParIntProcess.Value29; // Target Position FreshAir 2
      L     1;
      +I    ;
      T     "MAL1S021Par".Par.ParIntProcess.Value29; // Target Position FreshAir 2
      SPA   e615;
dez1: NOP   0;
      U     "MAL1S021Par".Par.FlagProcess.Inf06; // FreshAir Flap CLOSE
      U     "SYS_Scan0_Tick1min";
      SPBN  e615;
      L     "MAL1S021Par".Par.ParIntProcess.Value29; // Target Position FreshAir 2
      L     "MAL1S021Par".StepAct.PosFreshAirFlapBasic; // limit min
      <=I   ;
      SPB   e615;
      L     "MAL1S021Par".Par.ParIntProcess.Value29; // Target Position FreshAir 2
      L     1;
      -I    ;
      T     "MAL1S021Par".Par.ParIntProcess.Value29; // Target Position FreshAir 2
      SPA   e615;

sum1: NOP   0;
      L     "MAL1S021Par".StepAct.PosFreshAirFlapBasic;
      T     "MAL1S021Par".Par.ParIntProcess.Value29; // Target Position FreshAir 2
      SPA   e615;

e615: NOP   0;

NETWORK
TITLE =ASW_6080: Processtime Germinating
//      CALL  "SSA_MH_ProcessTime_Fct" , DB1017
//       InfDataReady :="MAL1S017".ToASW.InfDataReady
//       ProzessActive:="MAL1S017Par".Par.FlagProcess.ProcessActive
//       InStartTime  :="MAL1S017Par".Prozesstime.Starttime
//       OutStartTime :="MAL1S017Par".Prozesstime.Starttime
//       ProcessTime  :="MAL1S017Par".Prozesstime
//
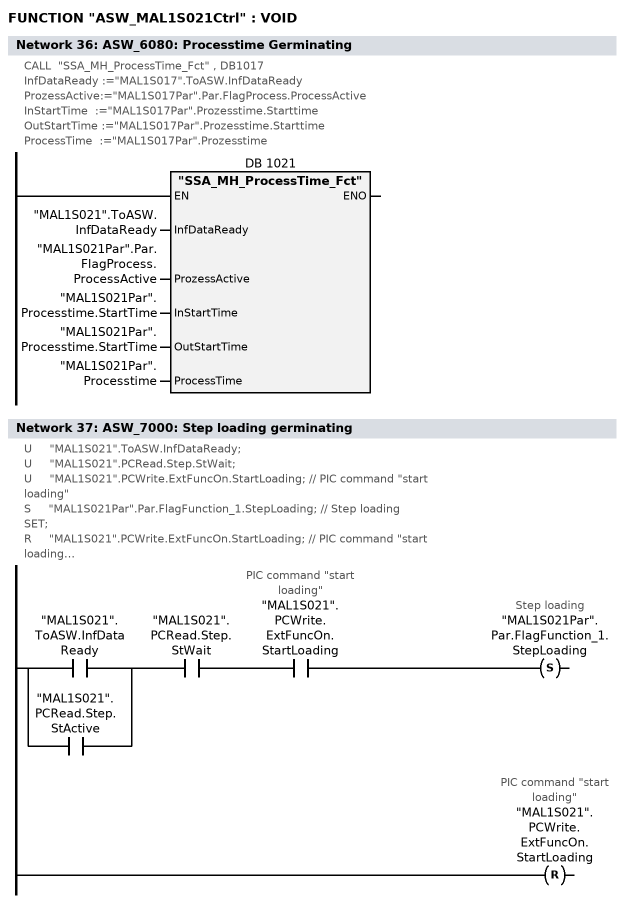
      CALL "SSA_MH_ProcessTime_Fct" , DB  1021 (
           InfDataReady             := "MAL1S021".ToASW.InfDataReady,
           ProzessActive            := "MAL1S021Par".Par.FlagProcess.ProcessActive,
           InStartTime              := "MAL1S021Par".Processtime.StartTime,
           OutStartTime             := "MAL1S021Par".Processtime.StartTime,
           ProcessTime              := "MAL1S021Par".Processtime);

NETWORK
TITLE =ASW_7000: Step loading germinating
//      U     "MAL1S021".ToASW.InfDataReady;
//      U     "MAL1S021".PCRead.Step.StWait;
//      U     "MAL1S021".PCWrite.ExtFuncOn.StartLoading; // PIC command "start
//loading"
//      S     "MAL1S021Par".Par.FlagFunction_1.StepLoading; // Step loading
//      SET;
//      R     "MAL1S021".PCWrite.ExtFuncOn.StartLoading; // PIC command "start
//loading"
////
//
//      L     WinCoS_BIW01_09PLC1BIW01_02.Ma.OutPositionAngle;
//      L     3600; // 360,0°
//      >=I   ;
//      U     "MAL1S021".ToASW.InfDataReady;
//      U     "MAL1S021".PCRead.Step.StActive;
//      U     "MAL1S021Par".Par.FlagFunction_1.StepLoading; // Step loading
//      =     "MAL1S021Par".Par.FlagFunction_1.LoadFirstPartEnd;
//
//      U     "MAL1S021".ToASW.InfDataReady;
//      U     "MAL1S021".PCRead.Step.StActive;
//      U     "MAL1S021Par".Par.FlagFunction_1.StepLoading; // Step loading
//      SPBN  E700;
//      L     "MAL1S021Par".RecipeHeader.Loading.LiftingPositionRound_1;
//      T     "MAL1S021Par".Par.ParIntProcess.NextLevelLoading; // next level
//
//      U(    ;
//      L     WinCoS_BIW01_09PLC1BIW01_02.Ma.OutPositionAngle;
//      L     "MAL1S021Par".Par.ParIntProcess.NextLevelLoading; // next level
//      >=I   ;
//      )     ;
//      O     "MAL1S021Par".Par.FlagMachine_0.Speed2ndRound;
//      SPB   Rnd2;
//      L     "MAL1S021Par".RecipeHeader.Loading.LoadingLevelRound_1;
//      T     "MAL1S021Par".Par.MachineValue.SOLLWERT_HUBZUG1_HOEHE;
//      T     "MAL1S021Par".Par.MachineValue.SOLLWERT_HUBZUG2_HOEHE;
//
//      L     "MAL1S021Par".RecipeHeader.Loading.LoadingSpeed_1;
//      T     "MAL1S021Par".Par.MachineValue.SollwertFahrantrieb;
//
//      SPA   Rnd1;
//Rnd2: NOP   0;
//      L     "MAL1S021Par".RecipeHeader.Loading.LoadingLevelRound_2;
//      T     "MAL1S021Par".Par.MachineValue.SOLLWERT_HUBZUG1_HOEHE;
//      T     "MAL1S021Par".Par.MachineValue.SOLLWERT_HUBZUG2_HOEHE;
//      L     10;
//      T     WinCoS_BIW01_09PLC1BIW01_02.Ma.Par.ParTolPosition;
//
//      L     15; // 15Hz = Wendegeschwindigkeit
//      T     "MAL1S021Par".Par.MachineValue.SollwertFahrantrieb;
//
//// Sicherheitsbit; damit bei manueller Rückwärtsfahrt über die 346°-Marke, nicht
// mit Loading Speed_0 durch den gefüllten KK gefahren wird!!
//      SET   ;
//      S     "MAL1S021Par".Par.FlagMachine_0.Speed2ndRound;
//
//Rnd1: NOP   0;
//      U  M 50.0;
//      =  M 50.0;
//      L     "MAL1S021Par".Par.ParIntMachine.TargetPosTravDriveLoad; // 450 =
//endposition loading
//      T     WinCoS_BIW01_09PLC1BIW01_02.Ma.InPositionTarget;
//E700: NOP   0;



      U     "MAL1S021".ToASW.InfDataReady;
      O     "MAL1S021".PCRead.Step.StActive;
      U     "MAL1S021".PCRead.Step.StWait;
      U     "MAL1S021".PCWrite.ExtFuncOn.StartLoading; // PIC command "start loading"
      S     "MAL1S021Par".Par.FlagFunction_1.StepLoading; // Step loading
      SET   ;
      R     "MAL1S021".PCWrite.ExtFuncOn.StartLoading; // PIC command "start loading"
//
      NOP   0;


NETWORK
TITLE =Sub 7010: Germination loading finished
//      U     "MAL1S021".ToASW.InfDataReady;
//      U     "MAL1S021".PCRead.Step.StActive;
//
//      UN    "MAL1S021".ToASW.InfSameJobPrevSec;
//      UN    "MAL1S021".PCRead.Step.StEmptying; // steep 1
//      U     "MAL1S021".PCWrite.ExtFuncOn.FinishLoading; // PIC command "finish
//loading"
//      U     "MAL1S021Par".Par.FlagFunction_1.StepLoading; // Step loading
//      S     "MAL1S021Par".Par.FlagFunction_1.FinishLoading; // loading is finish
//ed start process germinating
//      R     "MAL1S021Par".Par.FlagFunction_1.StepLoading; // Step loading
//
//      U     "MAL1S021".PCWrite.ExtFuncOn.FinishLoading; // PIC command "finish l
//oading"
//      R     "MAL1S021".PCWrite.ExtFuncOn.FinishLoading; // PIC command "finish l
//oading"
//
//      U     "MAL1S021Par".Par.FlagFunction_1.StepLoading; // Step loading
//      UN    "MAL1S021Par".Par.FlagFunction_1.FinishLoading; // loading is
//finished start process germinating
//      SPBN  save;
//      L     WinCoS_BIW01_09PLC1BIW01_02.Ma.OutPositionLeft;
//      L     WinCoS_BIW01_09PLC1BIW01_02.Ma.OutPositionRight;
//      +I    ;
//      L     2;
//      /I    ;
//      T     "MAL1S021Par".Par.ParIntMachine.LastLoadingLevel; // saved loading
//value
//save: NOP   0;
//
//      U     "MAL1S021".PCRead.Step.StReady;
//      O     "MAL1S021".PCRead.Step.StActive;
//      U     "MAL1S021Par".Par.FlagFunction_1.FinishLoading; // loading is
//finished start process germinating
//      UN     "MAL1S021Par".Par.FlagFunction_1.StepLoading; // Step loading
//      R     "MAL1S021Par".Par.FlagMachine_0.Speed2ndRound;
//fin:  NOP   0;
//E701: NOP   0;
// Previous Section always the Sec.801
///
      L     "MAL1S021".ToSSW.InPrevSecDB;
      L     0;
      <>I   ;
      SPB   prev;
      L     801;
      T     "MAL1S021".ToSSW.InPrevSecDB;
prev: NOP   0;


      U     "MAL1S021".ToASW.InfDataReady;
      U     "MAL1S021".PCRead.Step.StActive;
      UN    "MAL1S021".PCRead.Step.StEmptying; //
      U     "MAL1S021".PCWrite.ExtFuncOn.FinishLoading; // PIC command "finish loading"
      U     "MAL1S021Par".Par.FlagFunction_1.StepLoading; // Step loading
      O(    ;
      UN    "MAL1S021".SecNom.Par1On.Cmd01; // With Loading
      UN    "MAL1S021".ToASW.InfSameBatchPrevSec;
      U     "MAL1S021".ToASW.InfDataReady;
      U     "MAL1S021".PCRead.Step.StActive;
      )     ;
      S     "MAL1S021Par".Par.FlagFunction_1.FinishLoading; // loading is finished start process germinating
      R     "MAL1S021Par".Par.FlagFunction_1.StepLoading; // Step loading

      U     "MAL1S021".PCWrite.ExtFuncOn.FinishLoading; // PIC command "finish loading"
      R     "MAL1S021".PCWrite.ExtFuncOn.FinishLoading; // PIC command "finish loading"


      U     "MAL1S021".PCRead.Step.StReady;
      O     "MAL1S021".PCRead.Step.StActive;
      U     "MAL1S021Par".Par.FlagFunction_1.FinishLoading; // loading is finished start process germinating
      UN    "MAL1S021Par".Par.FlagFunction_1.StepLoading; // Step loading
      R     "MAL1S021Par".Par.FlagMachine_0.Speed2ndRound;
      NOP   0;
      NOP   0;


NETWORK
TITLE =ASW_8000:  Step unloading germination


      U     "MAL1S021".ToASW.InfDataReady;
      U     "MAL1S021".PCRead.Step.StEmptying;
//====>BRT070310
      U(    ;
      O     "MAL1S021".ToASW.InfSameJobNextSec;
      O(    ;
      L     831; // Next Section: MAL1S031
      L     "MAL1S021".SecNom.HEADER.Kilning_vessel_1; // Target in recipe
      ==I   ;
      )     ;
      )     ;
//<====BRT070310
      UN    "MAL1S021Par".Par.FlagFunction_1.StepUnloading; // Step unloading
      UN    "MAL1S021Par".Par.FlagFunction_1.FinishUnloading;
      U     "MAL1S021Par".Par.FlagMachine_0.CouplingDischargFinished;
      U     "MAL1S021Par".Par.FlagMachine_0.WallUnCoupled;
//BRT070310 - Start Unloading Button vergessen
      U     "MAL1S021".PCWrite.ExtFuncOn.StartUnLoading; // PIC command "Start Unloading"
      S     "MAL1S021Par".Par.FlagFunction_1.StepUnloading; // Step unloading

//BRT070310 - Start Unloading Button vergessen
      U     "MAL1S021".PCWrite.ExtFuncOn.StartUnLoading; // PIC command "Start Unloading"
      R     "MAL1S021".PCWrite.ExtFuncOn.StartUnLoading; // PIC command "Start Unloading"

      U     "MAL1S021Par".Par.FlagFunction_1.StepUnloading; // Step unloading
      U     "MAL1S021Par".Par.FlagFunction_1.UnloadingStarted;
//====>BRT070310
      U(    ;
      O     "MAL1S021".ToASW.spare34; // infNextSectionFeeding
      O(    ;
      L     831; // Next Section: MAL1S031
      L     "MAL1S021".SecNom.HEADER.Kilning_vessel_1; // Target in recipe
      ==I   ;
      )     ;
      )     ;
//<====BRT070310
      =     "MAL1S021Par".Par.FlagFunction_0.InfReleaseUnloading; // from kiln

      U     "MAL1S021Par".Par.FlagFunction_1.StepUnloading; // Step unloading
      UN    "MAL1S021Par".Par.FlagFunction_1.UnloadingStarted;
      U     "G182M".A_2515_BZS22.StFalse; // backwall is not in down pos
      U     "G182M".A_2515_BZS23.StTrue; // backwall is in up pos  // JV030908
      U     "G187M".A_2511_KCL01I5.StTrue; // pushbutton drive fast fwd
      S     "MAL1S021Par".Par.FlagFunction_1.UnloadingStarted;
      FP    "MAL1S021Par".Par.FlagFunction_0.FlagUnloadingStartedFP; // JV030908
      =     "MAL1S021Par".Par.FlagFunction_0.ImpulseUnloadingStarted; // JV030908

      UN    "MAL1S021Par".Par.FlagFunction_1.UnloadingStarted;
      O     "MAL1S021Par".Par.FlagFunction_1.StepCleaning; // Step cleaning
      O     "MAL1S021Par".Par.FlagFunction_1.FinishCleaning;
      SPB   EN38;
//BRT250310      L     3600
      L     4000; //BRT250310 -> +2° Overlapping damit die Maschine sicher auf den Endschalter fährt!
      T     "G185M".A_2511_MXZ41MA.Ma.InPositionTarget; // target position unloading
      L     "MAL1S021Par".RecipeHeader.Unloading.UnLoadingSpeed_2; // JV 290808
      T     "MAL1S021Par".Par.ParIntProcess.CopyLoadindSpeed2; // JV 290808
EN38: NOP   0;




NETWORK
TITLE =ASW_8010:  Step unloading finished

// Verweilzeit auf dem Endschalter  =A_2111_BZS44.StTrue --> stop discharge side
//      L     S5T#5M                      // Verweilzeit auf dem Endschalter
//BRT140310      U     "G185M".A_2511_BZS44.StTrue // stop discharge side
      U     "G185M".A_2511_BZS46.StTrue; // stop endposition unloading
//BRT140310      U     "G184M".A_2515_BZS42.StTrue
      U     "G186M".A_2515_MXZ11MA.Ma.StStartedFwd;
//      SE    T    121
//====>BRT070410 - ohne Timer, um Restart der Wartezeit bei Unterbruch Transport zu verhindern!
      UN    "MAL1S021Par".Par.FlagFunction_0.Inf29; //Wartezeit 180s abgelaufen = 1
      U     "SYS_Scan0_Tick1s";
      SPBN  wait;
      L     "MAL1S021Par".Par.ParIntMachine.Value33; //aktuelle Wartezeit Maschine bei 100% Unloading-Position
      L     1;
      +I    ;
      T     "MAL1S021Par".Par.ParIntMachine.Value33; //aktuelle Wartezeit Maschine bei 100% Unloading-Position
wait: NOP   0;
      L     "MAL1S021Par".Par.ParIntMachine.Value33; //aktuelle Wartezeit Maschine bei 100% Unloading-Position
      L     180; // 180s
      >=I   ;
      =     "MAL1S021Par".Par.FlagFunction_0.Inf29; //Wartezeit 180s abgelaufen = 1
//<====BRT070410
//************************************************************************************************

      U     "MAL1S021".ToASW.InfDataReady;
      U     "MAL1S021".PCRead.Step.StEmptying;
//====>BRT070310
      U(    ;
      O     "MAL1S021".ToASW.InfSameJobNextSec;
      O(    ;
      L     831; // Next Section: MAL1S031
      L     "MAL1S021".SecNom.HEADER.Kilning_vessel_1; // Target in recipe
      ==I   ;
      )     ;
      )     ;
//<====BRT070310
      U     "MAL1S021Par".Par.FlagFunction_1.StepUnloading; // Step unloading
      UN    "MAL1S021Par".Par.FlagFunction_1.FinishUnloading;
      U     "MAL1S021Par".Par.FlagFunction_1.StepUnloading; // Step unloading
      U     "MAL1S021Par".Par.FlagFunction_1.UnloadingStarted;
//      U     T    121                    // Verweilzeit auf dem Endschalter ist abgelaufen
      U(    ;
      U     "MAL1S021Par".Par.FlagFunction_0.Inf29; //Wartezeit 180s abgelaufen = 1
      O     "MAL1S021".PCWrite.ExtFuncOn.FinishCleanSurface; // PIC command "Finish Unloading"
      )     ;
//------------ Confirmation is necessary to finish unloading **********************
      U(    ;
      L     "G185M".A_2511_MXZ41MA.Ma.OutPositionRel;
      L     950; //95%
      >I    ;
      )     ;
//      U     "MAL1S021".PCWrite.ExtFuncOn.FinishCleanSurface    // PIC command "Finish Unloading"
//************************************************************************************************
      R     "MAL1S021Par".Par.FlagFunction_1.StepUnloading; // Step unloading
      S     "MAL1S021Par".Par.FlagFunction_1.FinishUnloading;
      S     "MAL1S021Par".Par.FlagMachine_0.CmdTurnRevAfterUnloading;
      S     "MAL1S021Par".Par.FlagGen.Flag0024; // finished first unloading
      UN    "MAL1S021Par".Par.FlagMachine_0.CmdTurnRevAfterUnloading;
      SPB   EN39;
      L     3399;
      T     "G185M".A_2511_MXZ41MA.Ma.InPositionTarget; // target position
EN39: NOP   0;

NETWORK
TITLE =ASW_9000: Step cleaning germination box
//
      U     "MAL1S021".ToASW.InfDataReady;
      U(    ;
      U     "MAL1S021".PCRead.Step.StEmptied;
      O     "MAL1S021".PCRead.Step.StEmptying;
      )     ;
      U     "MAL1S021Par".Par.FlagFunction_1.FinishUnloading;
      U     "MAL1S021Par".Par.FlagMachine_0.CmdTurnRevAfterUnloading;
      UN    "MAL1S021Par".Par.FlagMachine_0.CleaningAfterUnloading;
      U(    ;
      L     "G185M".A_2511_MXZ41MA.Ma.OutPositionRel;
      L     956;
      <=I   ; // cleaning pos
      )     ;
      U     "G185M".A_2511_BZS46.StFalse; // stop endposition unloading //JV040310
      U     "MAL1S021Par".Par.FlagGen.Flag0024; // finished first unloading
      UN    "MAL1S021Par".Par.FlagGen.Flag0025; // wait pos. to unloading leftover
      UN    "MAL1S021Par".Par.FlagGen.Flag0026; // unloading leftover
      UN    "MAL1S021Par".Par.FlagGen.Flag0027; // finished unloading leftover
      O     "MAL1S021".PCWrite.ExtFuncOn.FinishCleanSurface; // PIC command "Finish Unloading"
      R     "MAL1S021Par".Par.FlagMachine_0.CmdTurnRevAfterUnloading;
      R     "MAL1S021Par".Par.FlagGen.Flag0024; // finished first unloading
      S     "MAL1S021Par".Par.FlagGen.Flag0025; // wait pos. to unloading leftover

//--- Zwischenschritt für Starten einer Restentladung ---
      U     "G187M".A_2511_KCL01I5.StTrue; // pushbutton drive fast fwd
      UN    "MAL1S021Par".Par.FlagGen.Flag0024; // finished first unloading
      U     "MAL1S021Par".Par.FlagGen.Flag0025; // wait pos. to unloading leftover
      UN    "MAL1S021Par".Par.FlagGen.Flag0026; // unloading leftover
      U(    ;
      U     "MAL1S021".PCRead.Step.StEmptied;
      O     "MAL1S021".PCRead.Step.StEmptying;
      )     ;
      U     "MAL1S021Par".Par.FlagFunction_1.FinishUnloading;
      UN    "MAL1S021Par".Par.FlagMachine_0.CmdTurnRevAfterUnloading;
      UN    "MAL1S021Par".Par.FlagMachine_0.CleaningAfterUnloading;
      U(    ;
      L     "G185M".A_2511_MXZ41MA.Ma.OutPositionRel;
      L     956;
      <=I   ; // cleaning pos
      )     ;
      U     "G185M".A_2511_BZS46.StFalse; // stop endposition unloading
      O     "MAL1S021".PCWrite.ExtFuncOn.FinishCleanSurface; // PIC command "Finish Unloading"
      R     "MAL1S021Par".Par.FlagMachine_0.CmdTurnRevAfterUnloading;
      R     "MAL1S021Par".Par.FlagGen.Flag0025; // wait pos. to unloading leftover
      S     "MAL1S021Par".Par.FlagGen.Flag0026; // unloading leftover

      UN    "MAL1S021Par".Par.FlagGen.Flag0026; // unloading leftover
      SPB   EN40;
      L     4000;
      T     "G185M".A_2511_MXZ41MA.Ma.InPositionTarget; // target position
EN40: NOP   0;

//--- Erreichen der Endposition nach Restentladung ---
      U     "G185M".A_2511_BZS46.StTrue; // stop endposition unloading
      U     "MAL1S021Par".Par.FlagFunction_1.FinishUnloading;
      U     "MAL1S021Par".Par.FlagGen.Flag0026; // unloading leftover
      U(    ;
      L     "G185M".A_2511_MXZ41MA.Ma.OutPositionRel;
      L     950; //95%
      >I    ;
      )     ;
      O     "MAL1S021".PCWrite.ExtFuncOn.FinishCleanSurface; // PIC command "Finish Unloading"
      R     "MAL1S021Par".Par.FlagGen.Flag0026; // unloading leftover
      S     "MAL1S021Par".Par.FlagGen.Flag0027; // finished unloading leftover
      S     "MAL1S021Par".Par.FlagMachine_0.CmdTurnRevAfterUnloading;

//********************************************************************************************

      U     "MAL1S021".ToASW.InfDataReady;
//====>BRT040310
      U(    ;
      U     "MAL1S021".PCRead.Step.StEmptied;
      O     "MAL1S021".PCRead.Step.StEmptying;
      )     ;
//<====BRT040310
      U     "MAL1S021Par".Par.FlagFunction_1.FinishUnloading;
      U     "MAL1S021Par".Par.FlagMachine_0.CmdTurnRevAfterUnloading;
      UN    "MAL1S021Par".Par.FlagMachine_0.CleaningAfterUnloading;
      U(    ;
      L     "G185M".A_2511_MXZ41MA.Ma.OutPositionRel;
      L     956;
      <=I   ; // cleaning pos
      )     ;
      U     "G185M".A_2511_BZS46.StFalse; // stop endposition unloading //JV040310
//====>BRT120510
      UN    "MAL1S021Par".Par.FlagGen.Flag0024; // finished first unloading
      UN    "MAL1S021Par".Par.FlagGen.Flag0025; // wait pos. to unloading leftover
      UN    "MAL1S021Par".Par.FlagGen.Flag0026; // unloading leftover
      U     "MAL1S021Par".Par.FlagGen.Flag0027; // finished unloading leftover
      O     "MAL1S021".PCWrite.ExtFuncOn.FinishCleanSurface; // PIC command "Finish Unloading"
      R     "MAL1S021Par".Par.FlagGen.Flag0027; // finished unloading leftover
//<====BRT120510
      R     "MAL1S021Par".Par.FlagMachine_0.CmdTurnRevAfterUnloading;
      R     "MAL1S021Par".Par.FlagFunction_1.FinishUnloading;
      S     "MAL1S021Par".Par.FlagMachine_0.CleaningAfterUnloading;
      S     "MAL1S021Par".Par.FlagFunction_1.StepCleaning; // Step cleaning

      SET   ;
      R     "MAL1S021".PCWrite.ExtFuncOn.FinishCleanSurface; // PIC command "Finish Unloading"

NETWORK
TITLE =ASW_9010: Cleaning Germination box finished
//



      U     "MAL1S021".ToASW.InfDataReady;
//====>BRT070310
      U(    ;
      U     "MAL1S021".PCRead.Step.StEmptied;
      O     "MAL1S021".PCRead.Step.StEmptying;
      )     ;
//<====BRT070310
      U     "MAL1S021Par".Par.FlagFunction_1.StepCleaning; // Step cleaning
      U     "G185M".A_2511_BZS44.StFalse; // stop discharge side
      U(    ;
      O     "MAL1S021".PCWrite.ExtFuncOn.FinishCleaning; // PIC command "cleaning finished"
//BRT140310      O     "G187M".A_2511_KCL01I4.InpTrue    // pushbutton "drive rev"
      O     "G187M".A_2511_KCL01I6.InpTrue; // pushbutton "drive rev fast"
      )     ;
      R     "MAL1S021Par".Par.FlagMachine_0.CleaningAfterUnloading;
      R     "MAL1S021Par".Par.FlagFunction_1.StepCleaning; // Step cleaning
      S     "MAL1S021Par".Par.FlagFunction_1.FinishCleaning;

      SET   ;
      R     "MAL1S021".PCWrite.ExtFuncOn.FinishCleaning; // PIC command "cleaning finished"

      U     "MAL1S021".PCRead.Step.StIdling;
//BRT140310      U     "G185M".A_2511_BZS46.StTrue // stop fan side (home pos)
      U     "G185M".A_2511_BZS44.StTrue; // stop zeroposition (home pos)
      U(    ; //dyk 081031 50 pulses
      L     "G185M".A_2511_MXZ41MA.IncCounter.InpActCount;
      L     50;
      <I    ;
      )     ;
      R     "MAL1S021Par".Par.FlagFunction_1.FinishCleaning;

      UN    "MAL1S021Par".Par.FlagFunction_1.FinishCleaning;
      SPB   EN41;
      L     0;
      T     "G185M".A_2511_MXZ41MA.Ma.InPositionTarget; // target position
//MW 2008.10.24
      L     "MAL1S021Par".RecipeHeader.Unloading.UnLoadingSpeed_2;
      T     "MAL1S021Par".Par.ParIntProcess.CopyLoadindSpeed2;
EN41: NOP   0;

NETWORK
TITLE =ASW_9080: Send section date to PIC after germination

      AUF   "MAL1S021";
      U     "MAL1S021".PCRead.Step.StEmptying;
      FP    "MAL1S021Par".Par.FlagProcess.FP_SendResultToPIC;
      SPBN  E908;
//

E908: NOP   0;
NETWORK
TITLE =ASW_10000: ILO functions

      U     "MAL1S021".SecAc.Sta1On.Inf08;
      =     "MAL1S021".Gr.All.Spare04;

// reset ILO with start unloading   JV080908    special on SALADIN BOXES
      U     "MAL1S021Par".Par.FlagFunction_0.ImpulseUnloadingStarted; // JV030908
      R     "MAL1S021".SecAc.Sta1On.Inf08;

//- Little help for PIC-People
      U     "MAL1S021".SecAc.Sta1On.Inf08;
      SPB   RSM;
      L     0;
      T     "MAL1S021Par".Ilo.Code_ILO_Funktion0; // FCM 21 LINE 1 SEC   GERM 5
RSM:  NOP   0;
//- Combination OLD and NEW ---
      U     "MAL1S021".SecAc.Sta1On.Inf08;
      SPBN  IFM;
      L     "MAL1S021Par".Ilo.ILOMode;
      L     100;
      *I    ;
      T     "MAL1S021Par".Ilo.Code_ILO_Funktion0;
IFM:  NOP   0;

//  no ILO-mode >> cmd manual off to all used groups and reset all flags
      U     "MAL1S021".SecAc.Sta1On.Inf08;
      FN    "MAL1S021Par".Ilo.Flag.EdgeILOModeOn; //BRT140310
//BRT140310      FN    DB909.DBX 3692.0
//      S     DB909.DBX 3006.0            // (ManOff)
//      R     DB909.DBX 3014.0
//      R     DB909.DBX 3018.1
//  Gr-cmd manual OFF
      S     "G009G".Gr.CmdManualOff; // GENERAL ELEMENTS GERM 5
      S     "G182M".Gr.CmdManualOff; // LIFTING DEVICE  GERM 5
      S     "G183M".Gr.CmdManualOff; // COUPLING DEVICE TURNER  GERM 5
      S     "G184M".Gr.CmdManualOff; // COUPLING DEVICE WALL  GERM 5
      S     "G185M".Gr.CmdManualOff; // TRAVELLING DRIVE  GERM 5
      S     "G186M".Gr.CmdManualOff; // HORIZONTAL AND LIFTING SCREW  GERM 5
      S     "G189M".Gr.CmdManualOff; // TURNING SCREWS  GERM 5
      S     "G190M".Gr.CmdManualOff; // FAN AND VALVE SRAY AIR  GERM 5
      S     "G191M".Gr.CmdManualOff; // FRESH AIR LOUVER  GERM 5
      S     "G192M".Gr.CmdManualOff; // EXHAUST AIR LOUVER  GERM 5
      S     "G197M".Gr.CmdManualOff; // COOLING / HEATING  GERM 5
//  RESET ADDITIONAL CMD`S
      R     "G182M".USW14; // ILO-cmd
      R     "G182M".USW15; // ILO-cmd
      R     "G183M".USW14; // ILO-cmd
      R     "G183M".USW15; // ILO-cmd
      R     "G184M".USW14; // ILO-cmd
      R     "G184M".USW15; // ILO-cmd
      R     "G185M".USW14; // ILO-cmd
      R     "G185M".USW15; // ILO-cmd
      R     "G186M".USW14; // ILO-cmd
      R     "G186M".USW15; // ILO-cmd
      R     "G189M".USW14; // ILO-cmd
      R     "G189M".USW15; // ILO-cmd
      R     "G190M".USW14; // ILO-cmd
      R     "G190M".USW15; // ILO-cmd
      R     "G191M".USW14; // ILO-cmd
      R     "G191M".USW15; // ILO-cmd
      R     "G192M".USW14; // ILO-cmd
      R     "G192M".USW15; // ILO-cmd
      R     "G197M".USW14; // ILO-cmd
      R     "G197M".USW15; // ILO-cmd

      U     "MAL1S021".SecAc.Sta1On.Inf08;
      SPB   RSM2;
      L     0;
      T     #tmpInt;
      CALL "SIEMENS_FILL" (
           BVAL                     := #tmpInt,
           RET_VAL                  := #tmpRET,
           BLK                      := "MAL1S021Par".Ilo);
RSM2: NOP   0;


      NOP   0;
// --- FCM 04 - Fans ---
      L     "MAL1S021Par".Ilo.ILOMode;
      L     4;
      <>I   ;
      SPB   IO4;
// man on
      U     "MAL1S021Par".Ilo.GrCMDManOn[1];
      S     "G190M".Gr.InManual; // FAN AND VALVE SRAY AIR  GERM 5
      S     "G191M".Gr.InManual; // FRESH AIR LOUVER  GERM 5
      S     "G192M".Gr.InManual; // EXHAUST AIR LOUVER  GERM 5
      R     "MAL1S021Par".Ilo.GrCMDManOn[1];
// man off
      U     "MAL1S021Par".Ilo.GrCMDManOff[1];
      S     "G190M".Gr.CmdManualOff; // FAN AND VALVE SRAY AIR  GERM 5
      R     "G190M".Gr.InManual; // FAN AND VALVE SRAY AIR  GERM 5
      R     "G190M".USW14; // ILO-cmd
      R     "G190M".USW15; // ILO-cmd
      S     "G191M".Gr.CmdManualOff; // FRESH AIR LOUVER  GERM 5
      R     "G191M".Gr.InManual; // FRESH AIR LOUVER  GERM 5
      R     "G191M".USW14; // ILO-cmd
      R     "G191M".USW15; // ILO-cmd
      S     "G192M".Gr.CmdManualOff; // EXHAUST AIR LOUVER  GERM 5
      R     "G192M".Gr.InManual; // EXHAUST AIR LOUVER  GERM 5
      R     "G192M".USW14; // ILO-cmd
      R     "G192M".USW15; // ILO-cmd
      R     "MAL1S021Par".Ilo.GrCMDManOff[1];
      R     "MAL1S021Par".Ilo.GrCMDManAdditional.Cmd1[1];
      R     "MAL1S021Par".Ilo.GrCMDManAdditional.Cmd2[1];
// man start
      U     "MAL1S021Par".Ilo.GrCMDManStart[1];
      S     "G190M".Gr.CmdOn; // FAN AND VALVE SRAY AIR  GERM 5
      S     "G190M".Gr.CmdContinue; // FAN AND VALVE SRAY AIR  GERM 5
      S     "G191M".Gr.CmdOn; // FRESH AIR LOUVER  GERM 5
      S     "G191M".Gr.CmdContinue; // FRESH AIR LOUVER  GERM 5
      S     "G192M".Gr.CmdOn; // EXHAUST AIR LOUVER  GERM 5
      S     "G192M".Gr.CmdContinue; // EXHAUST AIR LOUVER  GERM 5
      R     "MAL1S021Par".Ilo.GrCMDManStart[1];
      U     "MAL1S021Par".Ilo.GrCMDManStart[2];
      R     "MAL1S021Par".Ilo.GrCMDManStart[2];
// man stop
      U     "MAL1S021Par".Ilo.GrCMDManStop[1];
      S     "G190M".Gr.CmdOff; // FAN AND VALVE SRAY AIR  GERM 5
//BRT140310      S     "G190M".Gr.CmdOff           // FRESH AIR LOUVER  GERM 5
//BRT140310      S     "G190M".Gr.CmdOff           // EXHAUST AIR LOUVER  GERM 5
      R     "MAL1S021Par".Ilo.GrCMDManStop[1];
// man fault reset
//BRT140310      U     "MAL1S021Par".Ilo.GrCMDManOn[17]
      U     "MAL1S021Par".Ilo.GrCMDManFaultReset[1]; //BRT140310
      S     "G190M".Gr.CmdFaultReset; // FAN AND VALVE SRAY AIR  GERM 5
      S     "G191M".Gr.CmdFaultReset; // FRESH AIR LOUVER  GERM 5
      S     "G192M".Gr.CmdFaultReset; // EXHAUST AIR LOUVER  GERM 5
//BRT160310      R     "MAL1S021Par".Ilo.GrCMDManOn[17]
      R     "MAL1S021Par".Ilo.GrCMDManFaultReset[1]; //BRT160310
// target position
      UN    "G190M".Gr.InManual; // FAN AND VALVE SRAY AIR  GERM 5
      O(    ;
      L     "MAL1S021Par".Ilo.Code_ILO_Funktion0;
      L     400;
      <>I   ;
      )     ;
      SPB   F04a;
      L     "MAL1S021Par".Ilo.SetpointInt01[1];
      T     "MAL1S021Par".Par.ParIntProcess.Speed_ILO_Fan;
F04a: NOP   0;
//BRT140310 - Sollwert Frischluftklappen!
      UN    "G191M".Gr.InManual; // FRESH AIR LOUVER GERM 5
      O(    ;
      L     "MAL1S021Par".Ilo.Code_ILO_Funktion0;
      L     400;
      <>I   ;
      )     ;
      SPB   F04b;
      L     "MAL1S021Par".Ilo.SetpointInt02[1];
      T     "MAL1S021Par".Par.ParIntProcess.TarPos_ILO_FreshAir;
F04b: NOP   0;

IO4:  NOP   0;
      NOP   0;
// --- FCM 05 - Fans with target air temperature ---
      L     "MAL1S021Par".Ilo.ILOMode;
      L     5;
      <>I   ;
      SPB   IO5;
// man on
      U     "MAL1S021Par".Ilo.GrCMDManOn[1];
      S     "G190M".Gr.InManual; // FAN AND VALVE SRAY AIR  GERM 5
      S     "G191M".Gr.InManual; // FRESH AIR LOUVER  GERM 5
      S     "G192M".Gr.InManual; // EXHAUST AIR LOUVER GERM 5  //BRT140310
      S     "G197M".Gr.InManual; // COOLING / HEATING  GERM 5
      R     "MAL1S021Par".Ilo.GrCMDManOn[1];
// man off
      U     "MAL1S021Par".Ilo.GrCMDManOff[1];
      S     "G190M".Gr.CmdManualOff; // FAN AND VALVE SRAY AIR  GERM 5
      R     "G190M".Gr.InManual; // FAN AND VALVE SRAY AIR  GERM 5
      R     "G190M".USW14; // ILO-cmd
      R     "G190M".USW15; // ILO-cmd
      S     "G191M".Gr.CmdManualOff; // FRESH AIR LOUVER  GERM 5
      R     "G191M".Gr.InManual; // FRESH AIR LOUVER  GERM 5
      R     "G191M".USW14; // ILO-cmd
      R     "G191M".USW15; // ILO-cmd
      S     "G192M".Gr.CmdManualOff; // EXHAUST AIR LOUVER GERM 5  //BRT140310
      R     "G192M".Gr.InManual; // EXHAUST AIR LOUVER GERM 5  //BRT140310
      R     "G192M".USW14; // ILO-cmd                    //BRT140310
      R     "G192M".USW15; // ILO-cmd                    //BRT140310
      S     "G197M".Gr.CmdManualOff; // COOLING / HEATING  GERM 5
      R     "G197M".Gr.InManual; // COOLING / HEATING  GERM 5
      R     "G197M".USW14; // ILO-cmd
      R     "G197M".USW15; // ILO-cmd
      R     "MAL1S021Par".Ilo.GrCMDManOff[1];
      R     "MAL1S021Par".Ilo.GrCMDManAdditional.Cmd1[1];
      R     "MAL1S021Par".Ilo.GrCMDManAdditional.Cmd2[1];
// man start
      U     "MAL1S021Par".Ilo.GrCMDManStart[1];
      S     "G190M".Gr.CmdOn; // FAN AND VALVE SRAY AIR  GERM 5
      S     "G190M".Gr.CmdContinue; // FAN AND VALVE SRAY AIR  GERM 5
      S     "G191M".Gr.CmdOn; // FRESH AIR LOUVER  GERM 5
      S     "G191M".Gr.CmdContinue; // FRESH AIR LOUVER  GERM 5
      S     "G192M".Gr.CmdOn; // EXHAUST AIR LOUVER GERM 5   //BRT140310
      S     "G192M".Gr.CmdContinue; // EXHAUST AIR LOUVER GERM 5   //BRT140310
      S     "G197M".Gr.CmdOn; // COOLING / HEATING  GERM 5
      S     "G197M".Gr.CmdContinue; // COOLING / HEATING  GERM 5
      R     "MAL1S021Par".Ilo.GrCMDManStart[1];
      U     "MAL1S021Par".Ilo.GrCMDManStart[2];
      R     "MAL1S021Par".Ilo.GrCMDManStart[2];
// man stop
      U     "MAL1S021Par".Ilo.GrCMDManStop[1];
      S     "G190M".Gr.CmdOff; // FAN AND VALVE SRAY AIR  GERM 5
//BRT140310      S     "G191M".Gr.CmdOff           // FRESH AIR LOUVER  GERM 5
//BRT140310      S     "G192M".Gr.CmdOff           // EXHAUST AIR LOUVER GERM 5   //BRT140310
      S     "G197M".Gr.CmdOff; // COOLING / HEATING  GERM 5
      R     "MAL1S021Par".Ilo.GrCMDManStop[1];
// man fault reset
      U     "MAL1S021Par".Ilo.GrCMDManFaultReset[1];
      S     "G190M".Gr.CmdFaultReset; // FAN AND VALVE SRAY AIR  GERM 5
      S     "G191M".Gr.CmdFaultReset; // FRESH AIR LOUVER  GERM 5
      S     "G192M".Gr.CmdFaultReset; // EXHAUST AIR LOUVER GERM 5   //BRT140310
      S     "G197M".Gr.CmdFaultReset; // COOLING / HEATING  GERM 5
      R     "MAL1S021Par".Ilo.GrCMDManFaultReset[1];
// target position
      UN    "G197M".Gr.InManual; // COOLING / HEATING  GERM 5
      SPB   F05a;
      L     "MAL1S021Par".Ilo.SetpointInt02[1];
      T     "MAL1S021Par".Par.ParIntProcess.TargetTemperature_ILO;
F05a: NOP   0;
      UN    "G190M".Gr.InManual; // FAN AND VALVE SRAY AIR  GERM 5
      O(    ;
      L     "MAL1S021Par".Ilo.Code_ILO_Funktion0;
      L     500;
      <>I   ;
      )     ;
      SPB   F05b;
      L     "MAL1S021Par".Ilo.SetpointInt01[1];
      T     "MAL1S021Par".Par.ParIntProcess.Speed_ILO_Fan;
F05b: NOP   0;
//BRT070310 - Sollwert Frischluftklappen!
      UN    "G191M".Gr.InManual; // FRESH AIR LOUVER GERM 5
      O(    ;
      L     "MAL1S021Par".Ilo.Code_ILO_Funktion0;
      L     500;
      <>I   ;
      )     ;
      SPB   F05c;
      L     "MAL1S021Par".Ilo.SetpointInt03[1];
      T     "MAL1S021Par".Par.ParIntProcess.TarPos_ILO_FreshAir;
F05c: NOP   0;

IO5:  NOP   0;
      NOP   0;
// --- FCM 06 - Fresh air flap ---
      L     "MAL1S021Par".Ilo.ILOMode;
      L     6;
      <>I   ;
      SPB   IO6;
// man on
      U     "MAL1S021Par".Ilo.GrCMDManOn[1];
      S     "G191M".Gr.InManual; // FRESH AIR LOUVER  GERM 5
//      R     DB909.DBX 3032.0
// man off
      U     "MAL1S021Par".Ilo.GrCMDManOff[1];
      S     "G191M".Gr.CmdManualOff; // FRESH AIR LOUVER  GERM 5
      R     "G191M".Gr.InManual; // FRESH AIR LOUVER  GERM 5
      R     "G191M".USW14; // ILO-cmd
      R     "G191M".USW15; // ILO-cmd
      R     "MAL1S021Par".Ilo.GrCMDManOff[1];
      R     "MAL1S021Par".Ilo.GrCMDManAdditional.Cmd1[1];
      R     "MAL1S021Par".Ilo.GrCMDManAdditional.Cmd2[1];
// man start
      U     "MAL1S021Par".Ilo.GrCMDManStart[1];
      S     "G191M".Gr.CmdOn; // FRESH AIR LOUVER  GERM 5
      S     "G191M".Gr.CmdContinue; // FRESH AIR LOUVER  GERM 5
      R     "MAL1S021Par".Ilo.GrCMDManStart[1];
      U     "MAL1S021Par".Ilo.GrCMDManStart[2];
      R     "MAL1S021Par".Ilo.GrCMDManStart[2];

      U     "MAL1S021Par".Ilo.GrCMDManOn[1];
      R     "MAL1S021Par".Ilo.GrCMDManOn[1];
// man stop
      U     "MAL1S021Par".Ilo.GrCMDManStop[1];
      S     "G191M".Gr.CmdOff; // FRESH AIR LOUVER  GERM 5
      R     "MAL1S021Par".Ilo.GrCMDManStop[1];
// man fault reset
//BRT140310      U     "MAL1S021Par".Ilo.GrCMDManOn[17]
      U     "MAL1S021Par".Ilo.GrCMDManFaultReset[1]; //BRT140310
      S     "G191M".Gr.CmdFaultReset; // FRESH AIR LOUVER  GERM 5
      R     "MAL1S021Par".Ilo.GrCMDManOn[17];
// moving direction

// target position
      UN    "G191M".Gr.InManual; // FRESH AIR LOUVER  GERM 5
      SPB   F06b;
      L     "MAL1S021Par".Ilo.SetpointInt01[1];
      T     "MAL1S021Par".Par.ParIntProcess.TarPos_ILO_FreshAir;
F06b: NOP   0;

IO6:  NOP   0;
      NOP   0;
// --- FCM 09 - Floor drives ---
      L     "MAL1S021Par".Ilo.ILOMode;
      L     9;
      <>I   ;
      SPB   IO9;
// man on
      U     "MAL1S021Par".Ilo.GrCMDManOn[1];
      S     "G009G".Gr.InManual; // GENERAL ELEMENTS GERM 5
      S     "G185M".Gr.InManual; // TRAVELLING DRIVE  GERM 5
      S     "G189M".Gr.InManual; // TURNING SCREWS  GERM 5
      R     "MAL1S021Par".Ilo.GrCMDManOn[1];
// man off
      U     "MAL1S021Par".Ilo.GrCMDManOff[1];
      S     "G009G".Gr.CmdManualOff; // GENERAL ELEMENTS GERM 5
      R     "G009G".Gr.InManual; // GENERAL ELEMENTS GERM 5
      S     "G185M".Gr.CmdManualOff; // TRAVELLING DRIVE  GERM 5
      R     "G185M".Gr.InManual; // TRAVELLING DRIVE  GERM 5
      R     "G185M".USW14; // ILO-cmd
      R     "G185M".USW15; // ILO-cmd
      S     "G189M".Gr.CmdManualOff; // TURNING SCREWS  GERM 5
      R     "G189M".Gr.InManual; // TURNING SCREWS  GERM 5
      R     "G189M".USW14; // ILO-cmd
      R     "G189M".USW15; // ILO-cmd
      R     "MAL1S021Par".Ilo.GrCMDManOff[1];
      R     "MAL1S021Par".Ilo.GrCMDManAdditional.Cmd1[1];
      R     "MAL1S021Par".Ilo.GrCMDManAdditional.Cmd2[1];
// man start
      U     "MAL1S021Par".Ilo.GrCMDManStart[1];
      S     "G009G".Gr.CmdOn; // GENERAL ELEMENTS GERM 5
      S     "G009G".Gr.CmdContinue; // GENERAL ELEMENTS GERM 5
      S     "G185M".Gr.CmdOn; // TRAVELLING DRIVE  GERM 5
      S     "G185M".Gr.CmdContinue; // TRAVELLING DRIVE  GERM 5
      S     "G189M".Gr.CmdOn; // TURNING SCREWS  GERM 5
      S     "G189M".Gr.CmdContinue; // TURNING SCREWS  GERM 5
      U     "MAL1S021Par".Ilo.GrCMDManStart[1];
      R     "MAL1S021Par".Ilo.GrCMDManStart[1];
      U     "MAL1S021Par".Ilo.GrCMDManStart[2];
      R     "MAL1S021Par".Ilo.GrCMDManStart[2];
// man stop
      U     "MAL1S021Par".Ilo.GrCMDManStop[1];
//====>BRT140310 - vom "Man Off" rauskopiert nach "Man Stop" + BZS44/46 ausgetauscht!
      O(    ;
      U(    ;
      U     "G185M".A_2511_BZS46.StTrue; // stop discharge side
      O     "G185M".A_2511_BZS46.InpTrue;
      U     "G185M".Gr.InManual;
      U     "G185M".USW14; // ILO-cmd run fwd
      )     ;
      O(    ;
      U     "G185M".A_2511_BZS44.StTrue; // stop fan side
      O     "G185M".A_2511_BZS44.InpTrue; // stop fan side
      U     "G185M".Gr.InManual;
      U     "G185M".USW15; // ILO-cmd run rev
      )     ;
      U(    ;
      L     "MAL1S021Par".Ilo.ILOMode;
//BRT140310      L     8
      L     9; //BRT140310
      ==I   ;
      )     ;
      )     ;
//<====BRT140310
      S     "G185M".Gr.CmdOff; // TRAVELLING DRIVE  GERM 5
//BRT140310      S     "G189M".Gr.CmdOff           // TURNING SCREWS  GERM 5
      R     "G185M".USW14; // ILO-cmd run fwd  //BRT140310
      R     "G185M".USW15; // ILO-cmd run rev  //BRT140310
      R     "MAL1S021Par".Ilo.GrCMDManStop[1];
// man fault reset
      U     "MAL1S021Par".Ilo.GrCMDManFaultReset[1];
      S     "G009G".Gr.CmdFaultReset; // GENERAL ELEMENTS GERM 5
      S     "G185M".Gr.CmdFaultReset; // TRAVELLING DRIVE  GERM 5
      S     "G189M".Gr.CmdFaultReset; // TURNING SCREWS  GERM 5
      R     "MAL1S021Par".Ilo.GrCMDManFaultReset[1];
// manual direction
      UN    "G185M".Gr.InManual; // TRAVELLING DRIVE  GERM 5
      SPB   f092;
      U     "MAL1S021Par".Ilo.GrCMDManAdditional.Cmd1[1];
      =     "G185M".USW14; // ILO-cmd run fwd
      U     "MAL1S021Par".Ilo.GrCMDManAdditional.Cmd2[1];
      =     "G185M".USW15; // ILO-cmd run rev
// target position
      L     "MAL1S021Par".Ilo.SetpointInt01[1];
      T     "MAL1S021Par".Par.ParIntProcess.Speed_ILO_FloorRotating;
f092: NOP   0;


IO9:  NOP   0;
// --- FCM 10 - local operating on operating panels ---

